// TwinCAT 3 PLC project SFICrane
// ProgramVersion: 3.1.4023.0
// libraries:
//   Tc2_MC2, * (Beckhoff Automation GmbH)
//   Tc2_MC2_Drive, * (Beckhoff Automation GmbH)
//   Tc2_Standard, * (Beckhoff Automation GmbH)
//   Tc2_System, * (Beckhoff Automation GmbH)
//   Tc2_Utilities, * (Beckhoff Automation GmbH)
//   Tc3_Module, * (Beckhoff Automation GmbH)
//   VisuDialogs, * (System)
// project tree:
//   AXIS CONTROL/ G_AXIS1.TcGVL, G_AXIS2.TcGVL, G_AXIS3.TcGVL, G_AXIS4.TcGVL, G_Safety_AXIS4.TcGVL, P_AxisControl.TcPOU, ST_MC_CMD.TcDUT (not stored), ST_MC_ParametersAxis.TcDUT (not stored), ST_MC_Status.TcDUT
//   / GlobalTextList.TcGTLO, MAIN.TcPOU, PlcTask.TcTTO, Visualization Manager.TcVMO (not stored)
//   HMI/ HMI.TcVIS
//   INPUTS/Function Blocks/ FB_AnalogInputScaling.TcPOU (not stored), FB_JoystickInputScaling.TcPOU (not stored)
//   INPUTS/GVL/ G_Inputs.TcGVL (not stored), G_ScalingParameters.TcGVL, G_Sensors.TcGVL
//   INPUTS/ P_Inputs.TcPOU
//   INPUTS/Struct/ ST_AnalogInput.TcDUT, ST_AnalogInputScaling.TcDUT (not stored), ST_AnalogInputStatus.TcDUT (not stored), ST_JoystickInputScaling.TcDUT (not stored), ST_Parameters.TcDUT (not stored)
//   MACHINE CONTROL/ G_MachineControl.TcGVL, P_MachineControl.TcPOU
//   MACHINE CONTROL/KinematicFunctions2d/ cosd.TcPOU (not stored), FB_Forward.TcPOU, FB_Inverse.TcPOU, FB_WireLengthOnCraneFunction.TcPOU, G_InverseKinematics.TcGVL, rt_ceild.TcPOU (not stored), rt_floord.TcPOU (not stored), rt_remd.TcPOU (not stored)
//   OUTPUTS/ G_Outputs.TcGVL, P_Outputs.TcPOU (not stored)
//   StablePlatform/Function Blocks/ FB_AnalogInputScalingPlusMinus.TcPOU, FB_AnalogInputScaling_1.TcPOU, FB_AutoModeControl.TcPOU, FB_Clock.TcPOU, FB_CylinderMotionControl.TcPOU, FB_JoystickInputScaling_1.TcPOU (not stored), FB_LowpassFilter.TcPOU, FB_RampMotionGenerator.TcPOU, FB_ValveOutput.TcPOU (not stored), FB_WaveMotionGenerator.TcPOU, FB_WaveMotionGenerator_1.TcPOU
//   StablePlatform/Functions/ fPlatformAngleTheta1.TcPOU, F_deg2rad.TcPOU, F_rad2deg.TcPOU, F_PlatformAnglePos2CylPos.TcPOU, F_PlatformAngleVel2CylVel.TcPOU
//   StablePlatform/GVL/ G_StablePlatformIO.TcGVL, G_StablePlatformParameters.TcGVL, G_StablePlatformScaledIO.TcGVL
//   StablePlatform/ P_StablePlatform.TcPOU, StablePlatform.TcVIS
//   StablePlatform/Struct/ ST_AnalogInputScaling_1.TcDUT (not stored), ST_JoystickInputScaling_1.TcDUT (not stored), ST_ValveDeadBand.TcDUT (not stored), ST_ValveOutput.TcDUT (not stored)
// real-time tasks:
//   TASK PlcTask: cycle T#2ms, priority 20, ADS port 350
// motion (NC):
//   TASK NC-Task 1 SAF: cycle T#2ms, priority 4, ADS port 501
//   TASK NC-Task 1 SVB: cycle T#10ms, priority 8, ADS port 511
//   AXIS Axis 1 - Main boom Cylinder (id 1)
//     Velo: SlowManual=20, FastManual=100
//     OtherSettings: AllowMotionCmdToSlave=true
//     encoder EncType=8
//       EncPara: MaxCount=#x0036ee7f
//         SoftEndMinControl: Enable=true, Range=12
//         SoftEndMaxControl: Enable=true, Range=298
//     drive DrvType=9
//       DrvPara: MaxCount=#xffffffff, DriveControlDWord=#x00030000
//         Analog: VeloScale=6, TorqueSetpointScale=10, ScaleFactorActTorque=0.1
//         TimeComp: TaskDelayCycles=1
//     controller CtrType=1
//       CtrPara: PriorControlFactor=1
//         Observer: BandWidth=20
//   AXIS Axis 2 - Slew Motor (id 5)
//     General: UnitName=Degree
//     Dynamic: AccelerationMaximum=55000, DecelerationMaximum=55000, Acceleration=30000, Deceleration=30000, Jerk=55000
//     Velo: SlowManual=200, FastManual=1000, Maximum=6000
//     OtherSettings: AllowMotionCmdToSlave=true, PulseDistancePos=100, PulseDistanceNeg=100
//     encoder EncType=8
//       EncPara: MaxCount=#xffffffff
//         SoftEndMinControl: Enable=true, Range=-32870
//         SoftEndMaxControl: Enable=true, Range=32800
//     drive DrvType=9
//       DrvPara: MaxCount=#xffffffff, DriveControlDWord=#x00030000
//         Analog: VeloReferenz=5000, VeloScale=6, TorqueSetpointScale=10, ScaleFactorActTorque=0.1
//         TimeComp: TaskDelayCycles=1
//     controller CtrType=1
//       CtrPara: PriorControlFactor=1
//         PosDiffControl: Range=20
//         Observer: BandWidth=20
//   AXIS Axis 3 - Knuckle boom Cylinder (id 3)
//     Velo: SlowManual=20, FastManual=100
//     OtherSettings: AllowMotionCmdToSlave=true
//     encoder EncType=8
//       EncPara: MaxCount=#x0036ee7f
//         SoftEndMinControl: Enable=true, Range=12
//         SoftEndMaxControl: Enable=true, Range=248
//     drive DrvType=9
//       DrvPara: MaxCount=#xffffffff, DriveControlDWord=#x00030000
//         Analog: VeloScale=6, TorqueSetpointScale=10, ScaleFactorActTorque=0.1
//         TimeComp: TaskDelayCycles=1
//     controller CtrType=1
//       CtrPara: PriorControlFactor=1
//         Observer: BandWidth=20
//   AXIS Axis 4 - Winch Motor (id 4)
//     General: UnitName=°
//     Dynamic: AccelerationMaximum=48322.755, DecelerationMaximum=48322.755, Acceleration=8053.79, Deceleration=8053.79, Jerk=24161.4
//     Velo: RefSearch=53.69195, RefSync=53.69195, SlowManual=268.45975, FastManual=1610.7585, Fast=5369.195
//     OtherSettings: AllowMotionCmdToSlave=true
//     encoder EncType=19
//       EncPara: ScaleFactorNumerator=60, ScaleFactorDenominator=1048576, MaxCount=#xffffffff
//     drive DrvType=16
//       DrvPara: MaxCount=#xffffffff, DriveControlDWord=#x00020000
//         Analog: VeloReferenz=5906.1145, VeloScale=32, TorqueSetpointScale=10, ScaleFactorActTorque=0.1
//         TimeComp: TaskDelayCycles=1
//     controller CtrType=1
//       CtrPara: PriorControlFactor=1
//         PosDiffControl: Enable=false
//         Observer: BandWidth=20
// I/O:
//   DEVICE Device 5 (EtherCAT), AmsNetId 5.107.189.26.6.1
//     Term 29 (EK1914) [EK1914, 2 Ch. Safety Input/Output 24V,  TwinSAFE]
//       modules: Module 1 (FSOE), Module 2 (DIO)
//     Drive 17 (IndraDrive MPB16/17) [IndraDrive MPB16/17]
//     Drive 22 (IndraDrive MPB20/21) [IndraDrive MPB20/21]
//     Drive 23 (IndraDrive MPB20/21) [IndraDrive MPB20/21]
//     Box 24 (AMI8000-0100) [AMI8000-0100 Servo motor 48 V DC, TwinSAFE]
//       modules: Module 1 (SAFETY)
//       startup 32785:21 := 0E01 // DRV Motor Settings / Commutation offset
//       startup 32786:19 := 0000 // DRV Brake Settings / Emergency application timeout
//       startup 32784:51 := 0A00 // DRV Amplifier Settings / Stand still window
//       startup 32784:19 := 2700 // DRV Amplifier Settings / Current loop proportional gain
//       startup 32784:18 := 1300 // DRV Amplifier Settings / Current loop integral time
//       startup 32784:21 := 1F010000 // DRV Amplifier Settings / Velocity loop proportional gain
//       startup 32784:20 := 96000000 // DRV Amplifier Settings / Velocity loop integral time
//   DEVICE Device 1 (EtherCAT), AmsNetId 5.107.189.26.2.1
//     Term 18 (EK1200) [EK1200-5000 EtherCAT Power supply (2A E-Bus)]
//       Term 20 (EL6910) [EL6910, TwinSAFE PLC]
//       Term 21 (EL1904) [EL1904, 4 Ch. Safety Input 24V, TwinSAFE]
//         modules: Module 1 (FSOES)
//       Term 25 (EL2008-0015) [EL2008-0015 8Ch. Dig. Output 24V DC, 0.35A, not short-circuit proof]
//       Term 26 (EK1110) [EK1110 EtherCAT extension]
//     Term 1 (EK1100) [EK1100 EtherCAT Coupler (2A E-Bus)]
//       Term 30 (EL3102) [EL3102 2Ch. Ana. Input +/-10V, Diff.]
//       Term 31 (EL3064) [EL3064 4Ch. Ana. Input 0-10V]
//       Term 32 (EL3124) [EL3124 4Ch. Ana. Input 4-20mA Diff.]
//       Term 33 (EL3154) [EL3154 4Ch. Ana. Input 4-20mA]
//       Term 34 (EL4122) [EL4122 2Ch. Ana. Output  4-20mA, 16bit]
//       Term 35 (EL3002) [EL3002 2Ch. Ana. Input +/-10V]
//       Term 36 (EL4132) [EL4132 2Ch. Ana. Output +/-10V, 16bit]
//       Term 37 (EL1859) [EL1859 8Ch. Dig. Input 24V, 3ms, 8Ch. Dig. Output 24V, 0.5A]
//       Term 35 (EL9011) [EL9011 End Terminal]
//     Term 27 (EK1818) [EK1818 EtherCAT IO-Coupler  (1A E-Bus, 8 Ch. Dig. In, 3ms, 4 Ch. Dig. Out 24V, 0,5A)]
//       Term 28 (EL3255) [EL3255 5Ch. potentiometer measurement with sensor supply]
//       Term 34 (EL9011) [EL9011 End Terminal]
// variable links:
//   Device 1 (EtherCAT) <-> Device 1 (EtherCAT)/Term 18 (EK1200)/Term 20 (EL6910)
//     Term 18 (EK1200)/Term 21 (EL1904)/Module 1 (FSOES)/TxPDO/FSOE <-> ConnectionOutputs/Message_4 RxPDO
//   Device 1 (EtherCAT) <-> Device 1 (EtherCAT)/Term 18 (EK1200)/Term 21 (EL1904)
//     Term 18 (EK1200)/Term 20 (EL6910)/ConnectionInputs/Message_4 TxPDO <-> Module 1 (FSOES)/RxPDO/FSOE
//   Device 1 (EtherCAT) <-> Device 5 (EtherCAT)/Box 24 (AMI8000-0100)
//     Term 18 (EK1200)/Term 20 (EL6910)/ConnectionInputs/Message_3 TxPDO <-> Module 1 (SAFETY)/SAFETY FSoE Connection 1 Receive Message/FSOE
//   Device 1 (EtherCAT) <-> Device 5 (EtherCAT)/Term 29 (EK1914)
//     Term 18 (EK1200)/Term 20 (EL6910)/ConnectionInputs/Message_5 TxPDO <-> Module 1 (FSOE)/Outputs/FSOE
//   Device 5 (EtherCAT) <-> Device 1 (EtherCAT)/Term 18 (EK1200)/Term 20 (EL6910)
//     Box 24 (AMI8000-0100)/Module 1 (SAFETY)/SAFETY FSoE Connection 1 Send Message/FSOE <-> ConnectionOutputs/Message_3 RxPDO
//     Term 29 (EK1914)/Module 1 (FSOE)/Inputs/FSOE <-> ConnectionOutputs/Message_5 RxPDO
//   NC-Task 1 SAF/Axes/Axis 1 - Main boom Cylinder <-> Device 5 (EtherCAT)/Drive 17 (IndraDrive MPB16/17)
//     Drive/Inputs/In/nDcOutputTime <-> InfoData/DcOutputShift
//     Drive/Inputs/In/nState1 <-> AT/Drive status word @bit 8
//     Drive/Inputs/In/nState2 <-> AT/Drive status word
//     Drive/Inputs/In/nState4 @bit 1 <-> WcState/InputToggle
//     Drive/Inputs/In/nState4 <-> WcState/WcState
//     Drive/Outputs/Out/nCtrl1 <-> MDT/Master control word @bit 8
//     Drive/Outputs/Out/nDataOut1 <-> MDT/Position command value
//     Enc/Inputs/In/nDataIn1 <-> AT/Position feedback value 1
//     Enc/Inputs/In/nDcInputTime <-> InfoData/DcInputShift
//     Enc/Inputs/In/nState4 @bit 1 <-> WcState/InputToggle
//     Enc/Inputs/In/nState4 <-> WcState/WcState
//   NC-Task 1 SAF/Axes/Axis 2 - Slew Motor <-> Device 5 (EtherCAT)/Drive 22 (IndraDrive MPB20/21)
//     Drive/Inputs/In/nDcOutputTime <-> InfoData/DcOutputShift
//     Drive/Inputs/In/nState1 <-> AT/Drive status word @bit 8
//     Drive/Inputs/In/nState2 <-> AT/Drive status word
//     Drive/Inputs/In/nState4 @bit 1 <-> WcState/InputToggle
//     Drive/Inputs/In/nState4 <-> WcState/WcState
//     Drive/Outputs/Out/nCtrl1 <-> MDT/Master control word @bit 8
//     Drive/Outputs/Out/nDataOut1 <-> MDT/Position command value
//     Enc/Inputs/In/nDataIn1 <-> AT/Position feedback value 1
//     Enc/Inputs/In/nDcInputTime <-> InfoData/DcInputShift
//     Enc/Inputs/In/nState4 @bit 1 <-> WcState/InputToggle
//     Enc/Inputs/In/nState4 <-> WcState/WcState
//   NC-Task 1 SAF/Axes/Axis 3 - Knuckle boom Cylinder <-> Device 5 (EtherCAT)/Drive 23 (IndraDrive MPB20/21)
//     Drive/Inputs/In/nDcOutputTime <-> InfoData/DcOutputShift
//     Drive/Inputs/In/nState1 <-> AT/Drive status word @bit 8
//     Drive/Inputs/In/nState2 <-> AT/Drive status word
//     Drive/Inputs/In/nState4 @bit 1 <-> WcState/InputToggle
//     Drive/Inputs/In/nState4 <-> WcState/WcState
//     Drive/Outputs/Out/nCtrl1 <-> MDT/Master control word @bit 8
//     Drive/Outputs/Out/nDataOut1 <-> MDT/Position command value
//     Enc/Inputs/In/nDataIn1 <-> AT/Position feedback value 1
//     Enc/Inputs/In/nDcInputTime <-> InfoData/DcInputShift
//     Enc/Inputs/In/nState4 @bit 1 <-> WcState/InputToggle
//     Enc/Inputs/In/nState4 <-> WcState/WcState
//   NC-Task 1 SAF/Axes/Axis 4 - Winch Motor <-> Device 5 (EtherCAT)/Box 24 (AMI8000-0100)
//     Drive/Inputs/In/nDataIn1 <-> DRV Following error actual value/Following error actual value
//     Drive/Inputs/In/nDcOutputTime <-> InfoData/DcOutputShift
//     Drive/Inputs/In/nState1 <-> DRV Statusword/Statusword
//     Drive/Inputs/In/nState2 <-> DRV Statusword/Statusword @bit 8
//     Drive/Inputs/In/nState4 @bit 1 <-> WcState/InputToggle
//     Drive/Inputs/In/nState4 <-> WcState/WcState
//     Drive/Outputs/Out/nCtrl1 <-> DRV Controlword/Controlword
//     Drive/Outputs/Out/nCtrl2 <-> DRV Controlword/Controlword @bit 8
//     Drive/Outputs/Out/nDataOut1 <-> DRV Target position/Target position
//     Drive/Outputs/Out/nDataOut2 <-> DRV Target velocity/Target velocity
//     Enc/Inputs/In/nDataIn1 <-> FB Position/Position
//     Enc/Inputs/In/nDcInputTime <-> InfoData/DcInputShift
//     Enc/Inputs/In/nState4 @bit 1 <-> WcState/InputToggle
//     Enc/Inputs/In/nState4 <-> WcState/WcState
//   SFICrane/SFICrane Instance <-> Device 1 (EtherCAT)/Term 1 (EK1100)/Term 31 (EL3064)
//     PlcTask Inputs/G_StablePlatformIO.npA <-> AI Standard Channel 1/Value
//     PlcTask Inputs/G_StablePlatformIO.npB <-> AI Standard Channel 2/Value
//     PlcTask Inputs/G_StablePlatformIO.npS <-> AI Standard Channel 3/Value
//   SFICrane/SFICrane Instance <-> Device 1 (EtherCAT)/Term 1 (EK1100)/Term 33 (EL3154)
//     PlcTask Inputs/G_StablePlatformIO.nSVFeedback <-> AI Standard Channel 1/Value
//   SFICrane/SFICrane Instance <-> Device 1 (EtherCAT)/Term 1 (EK1100)/Term 34 (EL4122)
//     PlcTask Outputs/G_StablePlatformIO.nSVControlSignal <-> Channel 1/Output
//   SFICrane/SFICrane Instance <-> Device 1 (EtherCAT)/Term 1 (EK1100)/Term 35 (EL3002)
//     PlcTask Inputs/G_StablePlatformIO.nPistonPosition <-> AI Standard Channel 1/Value
//     PlcTask Inputs/G_StablePlatformIO.nPistonVelocity <-> AI Standard Channel 2/Value
//   SFICrane/SFICrane Instance <-> Device 1 (EtherCAT)/Term 1 (EK1100)/Term 37 (EL1859)
//     PlcTask Outputs/G_StablePlatformIO.bSVEnable <-> Channel 14/Output
//   SFICrane/SFICrane Instance <-> Device 1 (EtherCAT)/Term 18 (EK1200)/Term 20 (EL6910)
//     PlcTask Inputs/G_Safety_AXIS4.ChA_STO_Active <-> StandardInputs/Standard Out Var 10
//     PlcTask Inputs/G_StablePlatformIO.bEMG_OK <-> StandardInputs/Standard Out Var 12
//     PlcTask Outputs/G_Safety_AXIS4.EMGRestart <-> StandardOutputs/Standard In Var 8
//     PlcTask Outputs/G_Safety_AXIS4.TwinSafeGroupComErrAck <-> StandardOutputs/Standard In Var 1
//     PlcTask Outputs/G_Safety_AXIS4.TwinSafeGroupRunStop <-> StandardOutputs/Standard In Var 2
//   SFICrane/SFICrane Instance <-> Device 1 (EtherCAT)/Term 18 (EK1200)/Term 25 (EL2008-0015)
//     PlcTask Outputs/G_Safety_AXIS4.bWinchMotor24vDisable <-> Channel 1/Output
//   SFICrane/SFICrane Instance <-> Device 1 (EtherCAT)/Term 27 (EK1818)
//     PlcTask Inputs/G_Inputs.bAutoModeSelector <-> Channel 4/Input
//     PlcTask Inputs/G_Inputs.bGreenButton <-> Channel 5/Input
//     PlcTask Inputs/G_Inputs.bJoystickLeftEnable <-> Channel 7/Input
//     PlcTask Inputs/G_Inputs.bJoystickRightEnable <-> Channel 8/Input
//     PlcTask Inputs/G_Inputs.bManualModeSelector <-> Channel 3/Input
//     PlcTask Inputs/G_Inputs.bRedButton <-> Channel 6/Input
//     PlcTask Inputs/G_StablePlatformIO.bModeSwitchOff <-> Channel 2/Input
//     PlcTask Outputs/G_Outputs.bGreenButtonLight <-> Channel 9/Output
//     PlcTask Outputs/G_Outputs.bRedButtonLight <-> Channel 10/Output
//   SFICrane/SFICrane Instance <-> Device 1 (EtherCAT)/Term 27 (EK1818)/Term 28 (EL3255)
//     PlcTask Inputs/G_Inputs.stJoyLX.nValue <-> AI Standard Channel 1/Value
//     PlcTask Inputs/G_Inputs.stJoyLX.stStatus <-> AI Standard Channel 1/Status
//     PlcTask Inputs/G_Inputs.stJoyLY.nValue <-> AI Standard Channel 2/Value
//     PlcTask Inputs/G_Inputs.stJoyLY.stStatus <-> AI Standard Channel 2/Status
//     PlcTask Inputs/G_Inputs.stJoyRX.nValue <-> AI Standard Channel 3/Value
//     PlcTask Inputs/G_Inputs.stJoyRX.stStatus <-> AI Standard Channel 3/Status
//     PlcTask Inputs/G_Inputs.stJoyRY.nValue <-> AI Standard Channel 4/Value
//     PlcTask Inputs/G_Inputs.stJoyRY.stStatus <-> AI Standard Channel 4/Status
//   SFICrane/SFICrane Instance <-> Device 5 (EtherCAT)/Term 29 (EK1914)
//     PlcTask Inputs/G_Inputs.bSafetyRelayRestartButton <-> Module 2 (DIO)/DIO Inputs/Input 0
//     PlcTask Outputs/G_Outputs.bSafetyRelayReset <-> Module 2 (DIO)/DIO Outputs/Output 0
//   SFICrane/SFICrane Instance <-> NC-Task 1 SAF/Axes/Axis 1 - Main boom Cylinder
//     PlcTask Inputs/G_AXIS1.BCAxis.NcToPlc <-> Outputs/ToPlc
//     PlcTask Inputs/G_MachineControl.fStrokeActuatorMain <-> Outputs/ToPlc/ActPos
//     PlcTask Outputs/G_AXIS1.BCAxis.PlcToNc <-> Inputs/FromPlc
//   SFICrane/SFICrane Instance <-> NC-Task 1 SAF/Axes/Axis 2 - Slew Motor
//     PlcTask Inputs/G_AXIS2.SJAxis.NcToPlc <-> Outputs/ToPlc
//     PlcTask Inputs/G_MachineControl.fSlewMotorAngle <-> Outputs/ToPlc/ActPos
//     PlcTask Outputs/G_AXIS2.SJAxis.PlcToNc <-> Inputs/FromPlc
//   SFICrane/SFICrane Instance <-> NC-Task 1 SAF/Axes/Axis 3 - Knuckle boom Cylinder
//     PlcTask Inputs/G_AXIS3.TCAxis.NcToPlc <-> Outputs/ToPlc
//     PlcTask Inputs/G_MachineControl.fStrokeActuatorKnuckle <-> Outputs/ToPlc/ActPos
//     PlcTask Outputs/G_AXIS3.TCAxis.PlcToNc <-> Inputs/FromPlc
//   SFICrane/SFICrane Instance <-> NC-Task 1 SAF/Axes/Axis 4 - Winch Motor
//     PlcTask Inputs/G_AXIS4.WMAxis.NcToPlc <-> Outputs/ToPlc
//     PlcTask Inputs/G_MachineControl.fWinchMotorAngleEncoder <-> Outputs/ToPlc/ActPos
//     PlcTask Outputs/G_AXIS4.WMAxis.PlcToNc <-> Inputs/FromPlc

CONFIGURATION SFICrane
    RESOURCE PLC ON TwinCAT3
        TASK PlcTask(INTERVAL := T#2ms, PRIORITY := 20);
        PROGRAM MAIN WITH PlcTask : MAIN;
    END_RESOURCE
END_CONFIGURATION

// ---- AXIS CONTROL/ST_MC_Status.TcDUT
TYPE ST_MC_Status :
STRUCT
	
Status			: BOOL;
Done			: BOOL;
Busy			: BOOL;
Error			: BOOL;
Active			: BOOL;
CmdAborted		: BOOL;
InVelocity		: BOOL;
ErrorID			: UDINT;
Enabled			: BOOL;

END_STRUCT
END_TYPE

// ---- INPUTS/Struct/ST_AnalogInput.TcDUT
TYPE ST_AnalogInput :
STRUCT
	stStatus AT %I* : ST_AnalogInputStatus;
	nValue AT %I* : INT;
END_STRUCT
END_TYPE

// ---- AXIS CONTROL/G_AXIS1.TcGVL
{attribute 'qualified_only'}
VAR_GLOBAL

//Axis1 Bottom Cylinder 'BC'
BCAxis : AXIS_REF;

//Motion Control Function Block Instant Variable 
fbBC_Reset				: MC_Reset;
fbBC_Power				: MC_Power;
fbBC_Stop				: MC_Stop;
fbBC_MoveVelocity		: MC_MoveVelocity;
fbBC_MoveAbs			: MC_MoveAbsolute;
fbBC_ExtSetDis			: MC_ExtSetPointGenDisable;
fbBC_ExtSetEnab			: MC_ExtSetPointGenEnable;
fbBC_ResetSet			: RS;

//Input: Command
bBC_ResetExe			: BOOL;
bBC_PowerEnCmd			: BOOL;
bBC_PowerEnPositive		: BOOL;
bBC_PowerEnNegative 	: BOOL;
bBC_StopExe				: BOOL;
bBC_MoveAbsExe			: BOOL;
bBC_ExtSetGenDisExe		: BOOL;
bBC_ExtSetGenEnaExe		: BOOL;
bBC_MoveAbsDone			: BOOL;

//Velocity commands structure
stBC_VelCmd				: ST_MC_CMD := (bExe := FALSE, lrVelocity := 100);//, EnuDirection := MC_Positive_Direction); 

//Variables/Parameters
lrBC_PowerOverride		: LREAL;
lrBC_MoveAbsPosition	: LREAL;
lrBC_MoveAbsVelocity	: LREAL;
lrBC_MoveAddPos			: LREAL;

// Status
stBC_Reset				: ST_MC_Status;
stBC_Power				: ST_MC_Status;
stBC_Stop				: ST_MC_Status;
stBC_MoveVelocity		: ST_MC_Status;
stBC_MoveAbs			: ST_MC_Status;
stBC_ExtSetDis			: ST_MC_Status;
stBC_ExtSetEnab			: ST_MC_Status;
stBC_ExtSetFeed			: ST_MC_Status;

END_VAR

// ---- AXIS CONTROL/G_AXIS2.TcGVL
{attribute 'qualified_only'}
VAR_GLOBAL

//Axis2 Slew Joint 'SJ'
SJAxis : AXIS_REF;

//Motion Control Function Block Instant Variable 
fbSJ_Reset				: MC_Reset;
fbSJ_Power				: MC_Power;
fbSJ_MoveVelocity		: MC_MoveVelocity;
fbSJ_Stop				: MC_Stop;

//Input: Command
bSJ_ResetExe			: BOOL;
bSJ_PowerEnCmd			: BOOL;
bSJ_PowerEnPositive		: BOOL;
bSJ_PowerEnNegative 	: BOOL;
bSJ_StopExe				: BOOL;

//Velocity commands structure
stSJ_VelCmd				: ST_MC_CMD := (bExe := FALSE, lrVelocity := 500, EnuDirection := MC_Positive_Direction); 

//Variables/Parameters
lrSJ_PowerOverride		: LREAL;

// Status
stSJ_Reset				: ST_MC_Status;
stSJ_Power				: ST_MC_Status;
stSJ_MoveVelocity		: ST_MC_Status;
stSJ_Stop				: ST_MC_Status;

END_VAR

// ---- AXIS CONTROL/G_AXIS3.TcGVL
{attribute 'qualified_only'}
VAR_GLOBAL

//Axis3 Top Cylinder 'TC'
TCAxis : AXIS_REF;

//Motion Control Function Block Instant Variable 
fbTC_Reset				: MC_Reset;
fbTC_Power				: MC_Power;
fbTC_MoveVelocity		: MC_MoveVelocity;
fbTC_Stop				: MC_Stop;
fbTC_MoveAbs			: MC_MoveAbsolute;
fbTC_ExtSetDis			: MC_ExtSetPointGenDisable;
fbTC_ExtSetEnab			: MC_ExtSetPointGenEnable;
fbTC_ResetSet			: RS;

//Input: Command
bTC_ResetExe			: BOOL;
bTC_PowerEnCmd			: BOOL;
bTC_PowerEnPositive		: BOOL;
bTC_PowerEnNegative 	: BOOL;
bTC_StopExe				: BOOL;
bTC_MoveAbsExe			: BOOL;
bTC_ExtSetGenDisExe		: BOOL;
bTC_ExtSetGenEnaExe		: BOOL;
bTC_MoveAbsDone			: BOOL;

//Velocity commands structure
stTC_VelCmd				: ST_MC_CMD := (bExe := FALSE, lrVelocity := 100, EnuDirection := MC_Positive_Direction); 

//Variables/Parameters
lrTC_PowerOverride		: LREAL;
lrTC_MoveAbsPosition	: LREAL;
lrTC_MoveAbsVelocity	: LREAL;
lrTC_MoveAddPos			: LREAL;

// Status
stTC_Reset				: ST_MC_Status;
stTC_Power				: ST_MC_Status;
stTC_MoveVelocity		: ST_MC_Status;
stTC_Stop				: ST_MC_Status;
stTC_MoveAbs			: ST_MC_Status;
stTC_ExtSetDis			: ST_MC_Status;
stTC_ExtSetEnab			: ST_MC_Status;
stTC_ExtSetFeed			: ST_MC_Status;

END_VAR

// ---- AXIS CONTROL/G_AXIS4.TcGVL
{attribute 'qualified_only'}
VAR_GLOBAL

//Axis4 Winch Motor 'WM'
WMAxis : AXIS_REF;

//Motion Control Function Block Instant Variable 
fbWM_Reset				: MC_Reset;
fbWM_Power				: MC_Power;
fbWM_MoveVelocity		: MC_MoveVelocity;
fbWM_Stop				: MC_Stop;
fbWM_MoveAbs			: MC_MoveAbsolute;
fbWM_ExtSetDis			: MC_ExtSetPointGenDisable;
fbWM_ExtSetEnab			: MC_ExtSetPointGenEnable;
fbWM_ResetSet			: RS;

//Input: Command
bWM_ResetExe			: BOOL;
bWM_PowerEnCmd			: BOOL;
bWM_PowerEnPositive		: BOOL;
bWM_PowerEnNegative 	: BOOL;
bWM_StopExe				: BOOL;
bWM_MoveAbsExe			: BOOL;
bWM_ExtSetGenDisExe		: BOOL;
bWM_ExtSetGenEnaExe		: BOOL;
bWM_MoveAbsDone			: BOOL;

//Velocity commands structure
stWM_VelCmd				: ST_MC_CMD := (bExe := FALSE, lrVelocity := 1000, EnuDirection := MC_Positive_Direction); 

//Variables/Parameters
lrWM_PowerOverride		: LREAL;
lrWM_MoveAbsPosition	: LREAL;
lrWM_MoveAbsVelocity	: LREAL;
lrWM_MoveAddPos			: LREAL;
lrWM_MoveSetPointVel	: LREAL;

//Direction
EnuMoveVelDirection		: MC_Direction;

// Status
stWM_Reset				: ST_MC_Status;
stWM_Power				: ST_MC_Status;
stWM_MoveVelocity		: ST_MC_Status;
stWM_Stop				: ST_MC_Status;
stWM_MoveAbs			: ST_MC_Status;
stWM_ExtSetDis			: ST_MC_Status;
stWM_ExtSetEnab			: ST_MC_Status;
stWM_ExtSetFeed			: ST_MC_Status;

END_VAR

// ---- AXIS CONTROL/G_Safety_AXIS4.TcGVL
{attribute 'qualified_only'}
VAR_GLOBAL
	
	bWinchMotor24vDisable 		AT %Q* : BOOL;
	TwinSafeGroupComErrAck 		AT %Q* : BOOL; 
	TwinSafeGroupRunStop 		AT %Q* : BOOL := FALSE; 
	ChA_STO_Enable 				AT %Q* : BOOL;
	ChA_STO_Active 				AT %I* : BOOL;  
	EMGRestart 					AT %Q* : BOOL; 
END_VAR

// ---- INPUTS/GVL/G_ScalingParameters.TcGVL
{attribute 'qualified_only'}
VAR_GLOBAL
	stParam : ST_Parameters;
END_VAR

// ---- INPUTS/GVL/G_Sensors.TcGVL
{attribute 'qualified_only'}
VAR_GLOBAL
	fJoystickLeftNormalizedY 		: LREAL;
	fJoystickLeftNormalizedX 		: LREAL;
	
	fJoystickRightNormalizedY 		: LREAL;
	fJoystickRightNormalizedX 		: LREAL;
	
	MCDirectionAxis1 : MC_Direction;
	MCDirectionAxis2 : MC_Direction;
	MCDirectionAxis3 : MC_Direction;
	MCDirectionAxis4 : MC_Direction;
	
		
END_VAR

// ---- MACHINE CONTROL/G_MachineControl.TcGVL
{attribute 'qualified_only'}
VAR_GLOBAL
	//Mode selector booleans
	bManualMode 			: BOOL;
	bAutoMode 				: BOOL;
	
	//Time variables
	fSampleTime				: LREAL := 0.002;
	fTimeSinceStart			: LREAL := 0.0;
	
	//Actuator position data
	fStrokeActuatorMain 	AT %I* : LREAL;
	fStrokeActuatorKnuckle 	AT %I* : LREAL;
	fSlewMotorAngle			AT %I* : LREAL;
	fWinchMotorAngleEncoder		AT %I* : LREAL;	
	fWinchAngle				: LREAL;
	fWinchMotorAngleRefDeg	: LREAL;
	
	//Positions from forward kinematics
	fCraneForwardX 			: LREAL;
	fCraneForwardY 			: LREAL;
	fTheta3Forward			: LREAL;
	fTheta4Forward			: LREAL;
	
	//Working parameters crane
	fWireLengthOnCrane		: LREAL;
	fPayloadHeightIni		: LREAL := 0.0;
	fWinchPitchRadiusLayer1 : LREAL := 0.0716;
	fWinchPitchRadiusLayer2 : LREAL := 0.0731;
	fWinchGearRatio 		: LREAL := 32;
	fWinchMotorAngleAbsRef	: LREAL;
	
	//Encoder values 
	fEncoderValue0Turns		: LREAL := 0.0;
	fEncoderValue5Turns		: LREAL := 0.0;
	fEncoderValueLayer2		: LREAL := 23666.0;
	fEncoderValueStartAuto	: LREAL;
	fTooltipYAutoStart		: LREAL;
	fRefPosPayloadAutoStart	: LREAL;
	fWinchMotorAngleRelRef	: LREAL;
	
	

END_VAR

// ---- MACHINE CONTROL/KinematicFunctions2d/G_InverseKinematics.TcGVL
{attribute 'qualified_only'}
VAR_GLOBAL
	fTooltipXCoordGlobalIni: LREAL := 2.8;
	fTooltipYCoordGlobalIni: LREAL := 2.2;
	
	fTheta1 : LREAL := 0;
	fAngleMainArmInverse :	LREAL;
	fAngleKnuckleArmInverse : LREAL;
	fStrokeActuatorMainInverse : LREAL;
	fStrokeActuatorKnuckleInverse : LREAL;
END_VAR

// ---- OUTPUTS/G_Outputs.TcGVL
{attribute 'qualified_only'}
VAR_GLOBAL
	// PLC Rack
	
	// RIO Rack
	// Digital Outputs
	bGreenButtonLight 			AT %Q* : BOOL;
	bRedButtonLight 			AT %Q* : BOOL;
	// Analog Outputs
	//stWinchValveOutput 		: ST_ValveOutput;
	//stCylValveOutput 			: ST_ValveOutput;
	bSafetyRelayReset		 	AT %Q* : BOOL;
END_VAR

// ---- StablePlatform/GVL/G_StablePlatformIO.TcGVL
{attribute 'qualified_only'}
VAR_GLOBAL
	bSVEnable AT %Q* : BOOL; 
	nSVControlSignal AT %Q* : INT; 
	//fJoyLeftX AT %I* : INT; 
	
	//bJoyLeftPushButton AT %I* : BOOL; 
	
	npA AT %I* : INT;
	npB AT %I* : INT;
	npS AT %I* : INT;
	
	nSVFeedback AT %I* : INT;
	
	bModeSwitchOff AT %I* : BOOL;
	
	nPistonPosition AT %I* : INT;
	nPistonVelocity AT %I* : INT;

	// TwinSAFE	
	bEMG_OK AT %I* : BOOL;
	
	// Visualizer HMI
	bEnable : BOOL;
	bModeSelector : BOOL;
	bManualMode : BOOL;
	bAutoMode : BOOL;
	bActivated : BOOL;
	
	// Stable Control
	bEnableFeedForward 		: BOOL := TRUE;
	fMaxValveFlow_lmin 		: LREAL := 45.0;
	bEnableFeedBackControl	: BOOL := TRUE;
	bEnableIntegralControl	: BOOL := FALSE;
	fProportionalGain		: LREAL := 25.0;
	fIntegralGain			: LREAL := 0.0;
	fMaxPosError_mm			: LREAL := 0.5;
	fCylVelRef_ms			: LREAL;
	fCylPosRef_m			: LREAL;
	fCylPos_m				: LREAL;
	bMotionModeSelector : BOOL;
	bStartMotionGenerator : BOOL;
	bRampMotionFullPeriode : BOOL;
	bRampMotionPos0_deg: LREAL := -2.0; 
	bRampMotionCylVel0_ms : LREAL := 0.0; 
	bRampMotionPositionSP_deg : LREAL := 0;
	bRampMotionVelocitySP_ms : LREAL := 0.025; 
	bRampMotiont0_s : LREAL := 1.0; 
	bRampMotiontRamp_s : LREAL := 1.0; 
	bRampMotiontHoldPos_s : LREAL := 2.0;

	fTime : LREAL;
	fWaveMotionAplitudeTheta0_deg : LREAL := -1.9; 
	WaveMotionFreq_rads : LREAL := 0.5;
	fWaveMotionOmega_degs : LREAL; 
	fWaveMotionTheta_deg : LREAL; 
	fAutoModeControlSignal :LREAL;
	
	fControlSignal : LREAL;
END_VAR

// ---- StablePlatform/GVL/G_StablePlatformParameters.TcGVL
{attribute 'qualified_only'}
VAR_GLOBAL
	stPressureSensorScaling400bar 	: ST_AnalogInputScaling := (fMaxInputValue := 32767.0, fMinInputValue := 0.0, fMaxOutputValue := 400.0, fMinOutputValue := 0.0);
	stJoystickInputScalingX 		: ST_JoystickInputScaling := (fMaxInputValue := 20625.0, fMinInputValue := 11800.0, fNeutralInputValue := 16265, fNeutralDeadband := 100.0, fMaxOutputValue := 1.0, fMinOutputValue := -1.0, fNeutralOutputValue := 0.0);
	stSVValveDeadBand 				: ST_ValveDeadBand := (fPosMax := 29490.0, fPosMin := 20950.0, fNegMin := 18250.0, fNegMax := 9830.0);
	stSVFeedbackScaling 			: ST_AnalogInputScaling := (fMaxInputValue := 32767.0, fMinInputValue := 0.0, fMaxOutputValue := 20.0, fMinOutputValue := 4.0);
	stPistonPos						: ST_AnalogInputScaling := (fMaxInputValue := 32767.0, fMinInputValue := -32767.0, fMaxOutputValue := 0.5, fMinOutputValue := 0.0);
	stPistonVel						: ST_AnalogInputScaling := (fMaxInputValue := 32767.0, fMinInputValue := -32767.0, fMaxOutputValue := 0.2, fMinOutputValue := -0.2);
	fMinLengthPlatformCylinder		: LREAL := 0.878;
	fCylLengthZeroAngle				: LREAL := 1.142;
	fLengthToCylinder				: LREAL := 0.500;
	fOffsetAngleDeg 				: LREAL := 55.4;
	fOffsetAngleRad					: LREAL := Tc2_Utilities.DEG_TO_RAD(fOffsetAngleDeg);
	fLengthA						: LREAL := 0.513; //Length from platform bearing to cylinder upper mount
	fLengthC						: LREAL := 1.353; //Length from platform bearing to cylinder lower mount
	fAngleOffsetDeg 				: LREAL := 0.0;
	fMaxControlSignal				: LREAL := 0.2; 
	fCutoffFreq 					: LREAL := 0.1;
	fDamping 						: LREAL := 0.707106781186547;
END_VAR

// ---- StablePlatform/GVL/G_StablePlatformScaledIO.TcGVL
{attribute 'qualified_only'}
VAR_GLOBAL
	bpA : LREAL; // 0..400bar
	bpB : LREAL; // 0..400bar
	bpS : LREAL; // 0..400bar
	fSVFeedback : LREAL; // 4..20 mA  | 0 = fault/off
	fJoystickNormalizedX : LREAL; // -1..0..1
	fPistonPosition : LREAL; //Piston position in meters
	fPistionPosFiltered : LREAL;
	fPistonVelocity : LREAL; //Piston velocity in meters/second
	fPlatformAngle	: LREAL; //Platform angle theta1 in radians
	fPlatformAngleDeg : LREAL;
END_VAR

// ---- MAIN.TcPOU
PROGRAM MAIN

VAR

END_VAR

P_Inputs();
P_MachineControl();
P_AxisControl();
P_Outputs();
P_StablePlatform();

END_PROGRAM

// ---- INPUTS/P_Inputs.TcPOU
PROGRAM P_Inputs
VAR
	fbJoystickLeftVert 					: FB_JoystickInputScaling;
	fbJoystickLeftHor 					: FB_JoystickInputScaling;
	
	fbJoystickRightVert 				: FB_JoystickInputScaling;
	fbJoystickRightHor 					: FB_JoystickInputScaling;
	
	bEnableJoystick : BOOL;
		
END_VAR

bEnableJoystick := NOT(G_StablePlatformIO.bManualMode);

fbJoystickLeftVert(
	bEnable := bEnableJoystick,
	nRawInput := G_Inputs.stJoyLY.nValue,
	stJoystickInputScaling := G_ScalingParameters.stParam.stJoystickInputScalingLeftY,
	fNormalizedOutput => G_Sensors.fJoystickLeftNormalizedY
);

IF G_Sensors.fJoystickLeftNormalizedY < 0 THEN
	G_Sensors.MCDirectionAxis3 := MC_Negative_Direction;
ELSIF G_Sensors.fJoystickLeftNormalizedY > 0 THEN
	G_Sensors.MCDirectionAxis3 := MC_Positive_Direction;	
END_IF

fbJoystickLeftHor(
	bEnable := bEnableJoystick,
	nRawInput := G_Inputs.stJoyLX.nValue,
	stJoystickInputScaling := G_ScalingParameters.stParam.stJoystickInputScalingLeftX,
	fNormalizedOutput => G_Sensors.fJoystickLeftNormalizedX
);

IF G_Sensors.fJoystickLeftNormalizedX < 0 THEN
	G_Sensors.MCDirectionAxis1 := MC_Positive_Direction;
ELSIF G_Sensors.fJoystickLeftNormalizedX > 0 THEN
	G_Sensors.MCDirectionAxis1 := MC_Negative_Direction;	
END_IF


fbJoystickRightVert(
	bEnable := bEnableJoystick,
	nRawInput := G_Inputs.stJoyRY.nValue,
	stJoystickInputScaling := G_ScalingParameters.stParam.stJoystickInputScalingRightY,
	fNormalizedOutput => G_Sensors.fJoystickRightNormalizedY
);

IF G_Sensors.fJoystickRightNormalizedY < 0 THEN
	G_Sensors.MCDirectionAxis4 := MC_Negative_Direction;
ELSIF G_Sensors.fJoystickRightNormalizedY > 0 THEN
	G_Sensors.MCDirectionAxis4 := MC_Positive_Direction;	
END_IF



fbJoystickRightHor(
	bEnable := bEnableJoystick,
	nRawInput := G_Inputs.stJoyRX.nValue,
	stJoystickInputScaling := G_ScalingParameters.stParam.stJoystickInputScalingRightX,
	fNormalizedOutput => G_Sensors.fJoystickRightNormalizedX
);

IF G_Sensors.fJoystickRightNormalizedX < 0 THEN
	G_Sensors.MCDirectionAxis2 := MC_Positive_Direction;
ELSIF G_Sensors.fJoystickRightNormalizedX > 0 THEN
	G_Sensors.MCDirectionAxis2 := MC_Negative_Direction;	
END_IF

END_PROGRAM

// ---- MACHINE CONTROL/P_MachineControl.TcPOU
PROGRAM P_MachineControl
VAR
	fbInverse					: FB_Inverse;
	fbForward					: FB_Forward;
	fbWireLengthOnCrane			: FB_WireLengthOnCraneFunction;
	fRefPosX					: LREAL := G_InverseKinematics.fTooltipXCoordGlobalIni;
	fRefPosY					: LREAL := G_InverseKinematics.fTooltipYCoordGlobalIni;	
	fRefPosPayload				: LREAL := G_MachineControl.fPayloadHeightIni;
	fWireLengthOutAutoStart		: LREAL;
	fWireLengthOut				: LREAL;
	fWireLengthOnCraneAutoStart	: LREAL;
	fWinchPitchRadius			: LREAL;
	fThetaWinch					: LREAL;
	bStartWave					: BOOL;
			
	
	
END_VAR

G_MachineControl.bManualMode := G_Inputs.bManualModeSelector;
G_MachineControl.bAutoMode := G_Inputs.bAutoModeSelector;
G_Safety_AXIS4.ChA_STO_Enable := G_Inputs.bManualModeSelector OR G_Inputs.bAutoModeSelector;

IF G_Inputs.bAutoModeSelector THEN
fRefPosX := fRefPosX + G_Sensors.fJoystickLeftNormalizedX*-0.0005;
fRefPosY := fRefPosY + G_Sensors.fJoystickLeftNormalizedY*0.0005;
fRefPosPayload := fRefPosPayload + G_Sensors.fJoystickRightNormalizedY*0.0002;
END_IF

bStartWave := NOT G_Inputs.bRedButton; //Red button is inverted, i.e. is active when not pushed

//Wave function used for testing
IF bStartWave THEN
	//Clock
	G_MachineControl.fTimeSinceStart := G_MachineControl.fTimeSinceStart + G_MachineControl.fSampleTime;
	G_InverseKinematics.fTheta1 := 0.012*SIN(2.5*G_MachineControl.fTimeSinceStart);
END_IF

(*
IF bStartWave THEN
	//Clock
	G_Work.fTimeSinceStart := G_Work.fTimeSinceStart + G_Work.fSampleTime;
	GVL_InverseKinematics.fTheta1 := G_StablePlatformParameters.fPlatformAngle;
END_IF
*)

fbInverse(
	fPtXd := fRefPosX, 
	fPtYd := fRefPosY, 
	//fTheta1 := G_InverseKinematics.fTheta1,
	fTheta1 := G_StablePlatformScaledIO.fPlatformAngleDeg*(PI/180),
	
	fTheta3 => G_InverseKinematics.fAngleMainArmInverse, 
	fTheta4 => G_InverseKinematics.fAngleKnuckleArmInverse,
	fStrokeActuatorMain => G_InverseKinematics.fStrokeActuatorMainInverse,
	fStrokeActuatorKnuckle => G_InverseKinematics.fStrokeActuatorKnuckleInverse,	
);

fbForward(
	fTheta1 := G_StablePlatformScaledIO.fPlatformAngle,
	fStrokeActuatorMain := (G_MachineControl.fStrokeActuatorMain+11),
	fStrokeActuatorKnuckle := (G_MachineControl.fStrokeActuatorKnuckle-7),
	x => G_MachineControl.fCraneForwardX,
	y => G_MachineControl.fCraneForwardY, 
	fTheta3 => G_MachineControl.fTheta3Forward,
	fTheta4 => G_MachineControl.fTheta4Forward,
);

fbWireLengthOnCrane(
	fTheta3 := G_MachineControl.fTheta3Forward,
	fTheta4 := G_MachineControl.fTheta4Forward,
	wireLengthOnCrane => G_MachineControl.fWireLengthOnCrane,
);

IF NOT (G_Inputs.bAutoModeSelector AND G_AXIS1.bBC_MoveAbsDone AND G_AXIS3.bTC_MoveAbsDone) THEN
	G_MachineControl.fEncoderValueStartAuto := G_MachineControl.fWinchMotorAngleEncoder;
	G_MachineControl.fRefPosPayloadAutoStart := G_MachineControl.fPayloadHeightIni;
	G_MachineControl.fTooltipYAutoStart := G_MachineControl.fCraneForwardY;	
	G_MachineControl.fWinchMotorAngleRelRef := G_MachineControl.fWinchMotorAngleRefDeg;
	fWireLengthOnCraneAutoStart := G_MachineControl.fWireLengthOnCrane;
END_IF

//fWireLengthOutAutoStart := fWireLengthOnCraneAutoStart + (G_MachineControl.fTooltipYAutoStart - G_MachineControl.fRefPosPayloadAutoStart);
fWireLengthOut := G_MachineControl.fWireLengthOnCrane + (G_MachineControl.fCraneForwardY - fRefPosPayload);


IF G_MachineControl.fWinchMotorAngleEncoder > G_MachineControl.fEncoderValueLayer2 THEN
	fWinchPitchRadius := G_MachineControl.fWinchPitchRadiusLayer2;
ELSE
	fWinchPitchRadius := G_MachineControl.fWinchPitchRadiusLayer1;
END_IF

fThetaWinch := (fWireLengthOut / fWinchPitchRadius);
G_MachineControl.fWinchMotorAngleRefDeg := fThetaWinch*G_MachineControl.fWinchGearRatio*180/PI;

IF NOT (G_Inputs.bAutoModeSelector AND G_AXIS1.bBC_MoveAbsDone AND G_AXIS3.bTC_MoveAbsDone) THEN
	G_MachineControl.fEncoderValueStartAuto := G_MachineControl.fWinchMotorAngleEncoder;
	
	G_MachineControl.fWinchMotorAngleRelRef := G_MachineControl.fWinchMotorAngleRefDeg;
END_IF

G_MachineControl.fWinchMotorAngleAbsRef := G_MachineControl.fEncoderValueStartAuto + G_MachineControl.fWinchMotorAngleRelRef - G_MachineControl.fWinchMotorAngleRefDeg;

END_PROGRAM

// ---- MACHINE CONTROL/KinematicFunctions2d/FB_Inverse.TcPOU
FUNCTION_BLOCK FB_Inverse
VAR_INPUT
	fPtXd: LREAL;
	fPtYd: LREAL;
	fTheta1: LREAL;
END_VAR
VAR_OUTPUT
	fStrokeActuatorMain: LREAL;
	fStrokeActuatorKnuckle: LREAL;
	fTheta3: LREAL;
	fTheta4: LREAL;
END_VAR
VAR
	h: LREAL;
	ThetaB: LREAL;
	ThetaB_tmp: LREAL;
	b_a_tmp: LREAL;
	a_tmp: LREAL;
	i0_cosd: cosd;
END_VAR


(* MATLAB Function: '<Root>/Inverse kinematics function' *)
(* clc; close all; clear; *)
(* MATLAB Function 'Inverse kinematics function': '<S1>:1' *)
(* Inputs *)
(* Desired global coordinates *)
(* fPtXd		= 0.75 + 1.5; *)
(* fPtYd		= 1.065 + 0.176; *)

(* %     fPtXd		= 0.75 + 0.716; *)
(* %  	fPtYd		= 1.065 + 0.705; *)
(* Platform constants *)
(* '<S1>:1:14' h0 = 1.0; *)
(* '<S1>:1:15' l0 = 0.75; *)
(* Crane constants *)
(* '<S1>:1:18' h1 = 1.334 + 0.065; *)
(* '<S1>:1:19' lm = 1.5; *)
(* '<S1>:1:20' lk = 1.158; *)
(* Calculate position of a2 as function of Theta1 *)
(* '<S1>:1:23' a2x = l0*cos(fTheta1) + h1*cos(fTheta1 + pi/2); *)
(* '<S1>:1:24' a2y = h0 + l0*sin(fTheta1) + h1*sin(fTheta1 + pi/2); *)
(* '<S1>:1:26' h = sqrt((fPtXd - a2x)^2 + (fPtYd - a2y)^2); *)
a_tmp := fPtXd - ((COS(fTheta1 + 1.5707963267948966) * 1.399) + (0.75 * COS(fTheta1)));
b_a_tmp := fPtYd - (((0.75 * SIN(fTheta1)) + 1.0) + (SIN(fTheta1 + 1.5707963267948966) * 1.399));
h := SQRT((a_tmp * a_tmp) + (b_a_tmp * b_a_tmp));
(* '<S1>:1:27' phi = atan((fPtYd - a2y) / (fPtXd - a2x)); *)
(* Calculate ThetaA and ThetaB *)
(* '<S1>:1:30' ThetaA = acos ((lm^2 + h^2 - lk^2) / (2*lm*h)); *)
(* '<S1>:1:31' ThetaB = acos ((lk^2 + lm^2 - h^2) / (2*lm*lk)); *)
ThetaB_tmp := h * h;
ThetaB := ACOS((3.5909639999999996 - ThetaB_tmp) / 3.4739999999999998);
(* '<S1>:1:33' fTheta3 = ThetaA + phi - fTheta1; *)
fTheta3 := (ACOS(((ThetaB_tmp + 2.25) - 1.3409639999999998) / (3.0 * h)) + ATAN(b_a_tmp / a_tmp)) - fTheta1;
(* '<S1>:1:34' fTheta4 = ThetaB - pi/2; *)
(* '<S1>:1:36' fTheta3deg = rad2deg(fTheta3); *)
(* '<S1>:1:37' fTheta4deg = rad2deg(fTheta4); *)
(* Crane constant parameters *)
(* '<S1>:1:40' fLengthP2PMainArm			= lm; *)
(* '<S1>:1:41' fLengthP2PKnuckleArm		= lk; *)
(* '<S1>:1:43' fLengthAMain				= 0.614; *)
(* '<S1>:1:44' fLengthBMain				= 0.571; *)
(* '<S1>:1:45' fMinLengthActuatorMain		= 0.691; *)
(* '<S1>:1:46' fMaxStrokeActuatorMain		= 0.290; *)
(* 0.320; *)
(* '<S1>:1:47' fMinStrokeActuatorMain		= 0.025; *)
(* '<S1>:1:49' fOffsetAngleDegMainAct		= 62.1; *)
(* '<S1>:1:51' fLengthAKnuckle				= 0.767; *)
(* '<S1>:1:52' fLengthBKnuckle				= 0.184; *)
(* '<S1>:1:53' fMinLengthActuatorKnuckle	= 0.633; *)
(* '<S1>:1:54' fMaxStrokeActuatorKnuckle	= 0.220; *)
(* 0.260; *)
(* '<S1>:1:55' fMinStrokeActuatorKnuckle   = 0.025; *)
(* '<S1>:1:57' fOffsetAngleDegKnuckleAct	= 86.3; *)
(* '<S1>:1:60' fAngleMainArmAct			= fTheta3deg + fOffsetAngleDegMainAct; *)
(* '<S1>:1:61' fAngleKnuckleArmAct         = fTheta4deg + fOffsetAngleDegKnuckleAct; *)
(* '<S1>:1:63' fLengthActuatorMain         = sqrt(fLengthAMain^2 + fLengthBMain^2 -(2*fLengthAMain*fLengthBMain*cosd(fAngleMainArmAct))); *)
(* '<S1>:1:64' fStrokeActuatorMain         = fLengthActuatorMain - fMinLengthActuatorMain; *)
a_tmp := (57.295779513082323 * fTheta3) + 62.1;
b_a_tmp := a_tmp;
i0_cosd(x := b_a_tmp);
(* Outport: '<Root>/fStrokeActuatorMain' incorporates:
 *  MATLAB Function: '<Root>/Inverse kinematics function' *)
fStrokeActuatorMain := SQRT(0.70303699999999991 - (0.70118799999999992 * b_a_tmp)) - 0.691;
(* MATLAB Function: '<Root>/Inverse kinematics function' *)
(* '<S1>:1:66' if fStrokeActuatorMain < fMinStrokeActuatorMain *)
b_a_tmp := a_tmp;
i0_cosd(x := b_a_tmp);

IF (SQRT(0.70303699999999991 - (0.70118799999999992 * b_a_tmp)) - 0.691) < 0.025 THEN 
    (* Outport: '<Root>/fStrokeActuatorMain' *)
    (* '<S1>:1:67' fStrokeActuatorMain = fMinStrokeActuatorMain; *)
    fStrokeActuatorMain := 0.025;
END_IF;

(* '<S1>:1:72' fLengthActuatorKnuckle         = sqrt(fLengthAKnuckle^2 + fLengthBKnuckle^2 -(2*fLengthAKnuckle*fLengthBKnuckle*cosd(fAngleKnuckleArmAct))); *)
(* '<S1>:1:73' fStrokeActuatorKnuckle         = fLengthActuatorKnuckle - fMinLengthActuatorKnuckle; *)
a_tmp := ((ThetaB - 1.5707963267948966) * 57.295779513082323) + 86.3;
b_a_tmp := a_tmp;
i0_cosd(x := b_a_tmp);
(* Outport: '<Root>/fStrokeActuatorKnuckle' incorporates:
 *  MATLAB Function: '<Root>/Inverse kinematics function' *)
fStrokeActuatorKnuckle := SQRT(0.62214500000000006 - (0.282256 * b_a_tmp)) - 0.633;
(* MATLAB Function: '<Root>/Inverse kinematics function' *)
(* '<S1>:1:75' if fStrokeActuatorKnuckle < fMinStrokeActuatorKnuckle *)
b_a_tmp := a_tmp;
i0_cosd(x := b_a_tmp);

IF (SQRT(0.62214500000000006 - (0.282256 * b_a_tmp)) - 0.633) < 0.025 THEN 
    (* Outport: '<Root>/fStrokeActuatorKnuckle' *)
    (* '<S1>:1:76' fStrokeActuatorKnuckle = fMinStrokeActuatorKnuckle; *)
    fStrokeActuatorKnuckle := 0.025;
END_IF;

(* Outport: '<Root>/fTheta4' incorporates:
 *  MATLAB Function: '<Root>/Inverse kinematics function' *)
fTheta4 := ThetaB - 1.5707963267948966;

END_FUNCTION_BLOCK

// ---- MACHINE CONTROL/KinematicFunctions2d/FB_Forward.TcPOU
FUNCTION_BLOCK FB_Forward
VAR_INPUT
	fTheta1: LREAL;
	fStrokeActuatorMain: LREAL;
	fStrokeActuatorKnuckle: LREAL;
END_VAR
VAR_OUTPUT
	x: LREAL;
	y: LREAL;
	fTheta3: LREAL;
	fTheta4: LREAL;
END_VAR
VAR
	x_tmp: LREAL;
	x_tmp_0: LREAL;
END_VAR


(* MATLAB Function: '<Root>/Forward kinematics actuator strokes' *)
(* Platform constants *)
(* MATLAB Function 'Forward kinematics actuator strokes': '<S1>:1' *)
(* '<S1>:1:4' fHeightPlatform = 1.402; *)
(* '<S1>:1:5' fHeightPlatformKing = 0.09; *)
(* '<S1>:1:6' fLengthPlatform = 1.30; *)
(* Crane and platform dimensions *)
(* Crane constant parameters *)
(* '<S1>:1:11' fHeightKingSlew             = 0.623; *)
(* '<S1>:1:12' fHeightSlewTop              = 0.711; *)
(* '<S1>:1:13' fLengthMainArm			    = 1.5; *)
(* '<S1>:1:14' fLengthKnuckleArm		    = 1.158; *)
(* '<S1>:1:16' fLengthAMain				= 0.614; *)
(* '<S1>:1:17' fLengthBMain				= 0.571; *)
(* '<S1>:1:18' fMinLengthActuatorMain		= 0.691; *)
(* '<S1>:1:19' fMaxStrokeActuatorMain		= 0.320; *)
(* '<S1>:1:21' fOffsetAngleDegMainAct		= 62.1; *)
(* '<S1>:1:22' fOffsetAngleRadMainAct		= deg2rad(fOffsetAngleDegMainAct); *)
(* '<S1>:1:24' fLengthAKnuckle				= 0.767; *)
(* '<S1>:1:25' fLengthBKnuckle				= 0.184; *)
(* '<S1>:1:26' fMinLengthActuatorKnuckle	= 0.633; *)
(* '<S1>:1:27' fMaxStrokeActuatorKnuckle	= 0.260; *)
(* '<S1>:1:29' fOffsetAngleDegKnuckleAct	= 86.3; *)
(* '<S1>:1:30' fOffsetAngleRadKnuckleAct	= deg2rad(fOffsetAngleDegKnuckleAct); *)
(* Calculating angles for main arm *)
(* '<S1>:1:33' fLengthActuatorMain = fStrokeActuatorMain + fMinLengthActuatorMain; *)
(* '<S1>:1:35' fAngleMainArmAct = acos((fLengthBMain^2 + fLengthAMain^2 - fLengthActuatorMain^2) / (2 * fLengthBMain * fLengthAMain)); *)
(* '<S1>:1:37' fTheta3 = fAngleMainArmAct - fOffsetAngleRadMainAct; *)
fTheta3 := ACOS((0.70303699999999991 - ((fStrokeActuatorMain/1000 + 0.691) * (fStrokeActuatorMain/1000 + 0.691))) / 0.70118799999999992) - 1.0838494654884787;
(* Calculating angles for knuckle arm *)
(* '<S1>:1:40' fLengthActuatorKnuckle = fStrokeActuatorKnuckle + fMinLengthActuatorKnuckle; *)
(* '<S1>:1:42' fAngleKnuckleArmAct = acos((fLengthBKnuckle^2 + fLengthAKnuckle^2 - fLengthActuatorKnuckle^2) / (2 * fLengthBKnuckle * fLengthAKnuckle)); *)
(* '<S1>:1:44' fTheta4 = fAngleKnuckleArmAct - fOffsetAngleRadKnuckleAct; *)
fTheta4 := ACOS((0.62214500000000006 - ((fStrokeActuatorKnuckle/1000 + 0.633) * (fStrokeActuatorKnuckle/1000 + 0.633))) / 0.282256) - 1.5062191444711064;

(* fAngleMainArmAct			= fTheta3deg + fOffsetAngleDegMainAct; *)
(* fAngleKnuckleArmAct         = fTheta4deg + fOffsetAngleDegKnuckleAct; *)

(* fLengthActuatorMain         = sqrt(fLengthAMain^2 + fLengthBMain^2 -(2*fLengthAMain*fLengthBMain*cosd(fAngleMainArmAct))); *)
(* fStrokeActuatorMain         = fLengthActuatorMain - fMinLengthActuatorMain; *)
(* if fStrokeActuatorMain < 0 *)
(* fStrokeActuatorMain = 0; *)
(* elseif fStrokeActuatorMain > fMaxStrokeActuatorMain *)
(* fMaxStrokeActuatorMain = fMaxStrokeActuatorMain; *)
(* end *)

(* fLengthActuatorKnuckle         = sqrt(fLengthAKnuckle^2 + fLengthBKnuckle^2 -(2*fLengthAKnuckle*fLengthBKnuckle*cosd(fAngleKnuckleArmAct))); *)
(* fStrokeActuatorKnuckle         = fLengthActuatorKnuckle - fMinLengthActuatorKnuckle; *)

(* if fStrokeActuatorKnuckle < 0 *)
(* fStrokeActuatorKnuckle = 0; *)
(* elseif fStrokeActuatorKnuckle > fMaxStrokeActuatorKnuckle *)
(* fMaxStrokeActuatorKnuckle = fMaxStrokeActuatorKnuckle; *)
(* end *)
(* '<S1>:1:71' fHeightMain                 = fHeightPlatformKing + fHeightKingSlew + fHeightSlewTop; *)
(* x = fLengthPlatform*cos(fTheta1) + fHeightMain*cos(fTheta1 + pi/2) + fLengthMainArm*cos(fTheta1 + fTheta3) + fLengthKnuckleArm * cos (fTheta1 + fTheta3 + fTheta4 - pi/2); *)
(* y = fHeightPlatform + fLengthPlatform*sin(fTheta1) + fHeightMain * sin(fTheta1 + pi/2) + fLengthMainArm *sin(fTheta1 + fTheta3) + fLengthKnuckleArm*sin(fTheta1 + fTheta3 + fTheta4 - pi/2); *)
(* '<S1>:1:76' x = fLengthPlatform*cos(fTheta1) + fHeightMain*cos(fTheta1 + pi/2) + fLengthMainArm*cos(fTheta1 + fTheta3) + fLengthKnuckleArm * cos (fTheta1 + fTheta3 + fTheta4 - pi/2); *)
(* '<S1>:1:77' y = fHeightPlatform + fLengthPlatform*sin(fTheta1) + fHeightMain * sin(fTheta1 + pi/2) + fLengthMainArm *sin(fTheta1 + fTheta3) + fLengthKnuckleArm*sin(fTheta1 + fTheta3 + fTheta4 - pi/2); *)
x_tmp := fTheta1 + fTheta3;
x_tmp_0 := (x_tmp + fTheta4) - 1.5707963267948966;
(* Outport: '<Root>/x' incorporates:
 *  MATLAB Function: '<Root>/Forward kinematics actuator strokes' *)
x := (((COS(fTheta1 + 1.5707963267948966) * 1.424) + (1.3 * COS(fTheta1))) + (COS(x_tmp) * 1.5)) + (COS(x_tmp_0) * 1.158);
(* Outport: '<Root>/y' incorporates:
 *  MATLAB Function: '<Root>/Forward kinematics actuator strokes' *)
y := ((((1.3 * SIN(fTheta1)) + 1.402) + (SIN(fTheta1 + 1.5707963267948966) * 1.424)) + (SIN(x_tmp) * 1.5)) + (SIN(x_tmp_0) * 1.158);

END_FUNCTION_BLOCK

// ---- MACHINE CONTROL/KinematicFunctions2d/FB_WireLengthOnCraneFunction.TcPOU
FUNCTION_BLOCK FB_WireLengthOnCraneFunction
VAR_INPUT
	fTheta3: LREAL;
	fTheta4: LREAL;
END_VAR
VAR_OUTPUT
	wireLengthOnCrane: LREAL;
END_VAR
VAR
	Ps1x: LREAL;
	Ps1y: LREAL;
	Ps2x: LREAL;
	Ps2y: LREAL;
	Ps3x: LREAL;
	Ps3y: LREAL;
	b_a: LREAL;
	d_a: LREAL;
	Ps1x_tmp: LREAL;
	Ps1x_tmp_0: LREAL;
	Ps3x_tmp_tmp: LREAL;
END_VAR


(* MATLAB Function: '<Root>/wireLengthOnCraneFunction1' *)
(* MATLAB Function 'wireLengthOnCraneFunction1': '<S1>:1' *)
(* '<S1>:1:3' lengthOrigoToWinch = 0.2199; *)
(* '<S1>:1:4' heightOrigoToWinch = 0.0895; *)
(* '<S1>:1:5' lengthOrigoToSheave1 = 0.2348; *)
(* '<S1>:1:6' heightOrigoToSheave1 = 0.060; *)
(* '<S1>:1:7' lengthOrigoToSheave2 = 1.520; *)
(* '<S1>:1:8' heigthOrigoToSheave2 = 0.095; *)
(* '<S1>:1:9' lengthMainArmToSheave3 = 0.2591; *)
(* '<S1>:1:10' lengthMainArmToSheave4 = 1.158; *)
(* '<S1>:1:11' offsetAngleSheave3deg = 49.7; *)
(* '<S1>:1:12' offsetAngleSheave3rad = deg2rad(offsetAngleSheave3deg); *)
(* '<S1>:1:13' offsetAngleSheave4deg = 90; *)
(* '<S1>:1:14' offsetAngleSheave4rad = deg2rad(offsetAngleSheave4deg); *)
(* '<S1>:1:16' lengthMainArm = 1.500; *)
(* '<S1>:1:17' pitchRadiusWinch = 0.0716; *)
(* '<S1>:1:18' pitchRadiusSheave = 0.034; *)
(* '<S1>:1:20' Pwx = -lengthOrigoToWinch; *)
(* '<S1>:1:21' Pwy = -heightOrigoToWinch; *)
(* '<S1>:1:22' Ps1x = lengthOrigoToSheave1 * cos(theta3) - heightOrigoToSheave1 * sin(theta3); *)
Ps1x_tmp := SIN(fTheta3);
Ps1x_tmp_0 := COS(fTheta3);
Ps1x := (0.2348 * Ps1x_tmp_0) - (0.06 * Ps1x_tmp);
(* '<S1>:1:23' Ps1y = lengthOrigoToSheave1 * sin(theta3) + heightOrigoToSheave1 * cos(theta3); *)
Ps1y := (0.2348 * Ps1x_tmp) + (0.06 * Ps1x_tmp_0);
(* '<S1>:1:24' Ps2x = lengthOrigoToSheave2 * cos(theta3) - heigthOrigoToSheave2 * sin(theta3); *)
Ps2x := (1.52 * Ps1x_tmp_0) - (0.095 * Ps1x_tmp);
(* '<S1>:1:25' Ps2y = lengthOrigoToSheave2 * sin(theta3) + heigthOrigoToSheave2 * cos(theta3); *)
Ps2y := (1.52 * Ps1x_tmp) + (0.095 * Ps1x_tmp_0);
(* '<S1>:1:26' Ps3x = lengthMainArm * cos(theta3) + lengthMainArmToSheave3 * cos(theta3 + theta4 - offsetAngleSheave3rad); *)
Ps3x_tmp_tmp := fTheta3 + fTheta4;
Ps3x := (COS(Ps3x_tmp_tmp - 0.86742863824118188) * 0.2591) + (1.5 * Ps1x_tmp_0);
(* '<S1>:1:27' Ps3y = lengthMainArm * sin(theta3) + lengthMainArmToSheave3 * sin(theta3 + theta4 - offsetAngleSheave3rad); *)
Ps3y := (SIN(Ps3x_tmp_tmp - 0.86742863824118188) * 0.2591) + (1.5 * Ps1x_tmp);
(* '<S1>:1:28' Ps4x = lengthMainArm * cos(theta3) + lengthMainArmToSheave4 * cos(theta3 + theta4 - offsetAngleSheave4rad); *)
(* '<S1>:1:29' Ps4y = lengthMainArm * sin(theta3) + lengthMainArmToSheave4 * sin(theta3 + theta4 - offsetAngleSheave4rad); *)
(* '<S1>:1:31' distanceWinchSheave1 =  sqrt((Ps1x - Pwx)^2 + (Ps1y - Pwy)^2); *)
Ps1x_tmp := SQRT(((Ps1x - -0.2199) * (Ps1x - -0.2199)) + ((Ps1y - -0.0895) * (Ps1y - -0.0895)));
(* distanceTwoPoints(Pwx, Pwy, Ps1x, Ps1y); *)
(* '<S1>:1:32' distanceSheave1Sheave2 = sqrt((Ps2x - Ps1x)^2 + (Ps2y - Ps1y)^2); *)
Ps1x_tmp_0 := Ps2x - Ps1x;
b_a := Ps2y - Ps1y;
Ps1x_tmp_0 := SQRT((Ps1x_tmp_0 * Ps1x_tmp_0) + (b_a * b_a));
(* distanceTwoPoints(Ps2x, Ps2y, Ps1x, Ps1y); *)
(* '<S1>:1:33' distanceSheave2Sheave3 = sqrt((Ps3x - Ps2x)^2 + (Ps3y - Ps2y)^2); *)
b_a := Ps3x - Ps2x;
d_a := Ps3y - Ps2y;
b_a := SQRT((b_a * b_a) + (d_a * d_a));
(* distanceTwoPoints(Ps2x, Ps2y, Ps3x, Ps3y); *)
(* '<S1>:1:34' distanceSheave3Sheave4 = sqrt((Ps4x - Ps3x)^2 + (Ps4y - Ps3y)^2); *)
d_a := ((COS(Ps3x_tmp_tmp - 1.5707963267948966) * 1.158) + (1.5 * COS(fTheta3))) - Ps3x;
Ps3x_tmp_tmp := ((SIN(Ps3x_tmp_tmp - 1.5707963267948966) * 1.158) + (1.5 * SIN(fTheta3))) - Ps3y;
d_a := SQRT((d_a * d_a) + (Ps3x_tmp_tmp * Ps3x_tmp_tmp));
(* Outport: '<Root>/wireLengthOnCrane' incorporates:
 *  MATLAB Function: '<Root>/wireLengthOnCraneFunction1' *)
(* distanceTwoPoints(Ps4x, Ps4y, Ps3x, Ps3y); *)
(* '<S1>:1:36' tangentLengthWinchSheave1 = sqrt(distanceWinchSheave1^2 -(pitchRadiusWinch -pitchRadiusSheave)^2); *)
(* tangentLengthFunction(distanceWinchSheave1, pitchRadiusWinch, pitchRadiusSheave); *)
(* '<S1>:1:37' tangentLengthSheave1Sheave2 = sqrt(distanceSheave1Sheave2^2 -(pitchRadiusSheave -pitchRadiusSheave)^2); *)
(* tangentLengthFunction(distanceSheave1Sheave2, pitchRadiusSheave, pitchRadiusSheave); *)
(* '<S1>:1:38' tangentLengthSheave2Sheave3 = sqrt(distanceSheave2Sheave3^2 -(pitchRadiusSheave -pitchRadiusSheave)^2); *)
(* tangentLengthFunction(distanceSheave2Sheave3, pitchRadiusSheave, pitchRadiusSheave); *)
(* '<S1>:1:39' tangentLengthSheave3Sheave4 = sqrt(distanceSheave3Sheave4^2 -(pitchRadiusSheave -pitchRadiusSheave)^2); *)
(* tangentLengthFunction(distanceSheave3Sheave4, pitchRadiusSheave, pitchRadiusSheave); *)
(* '<S1>:1:41' offsetAngleDeg = 113.6 + 9.9; *)
(* '<S1>:1:42' offsetAngleRad = deg2rad(offsetAngleDeg); *)
(* '<S1>:1:44' wrapAngle = offsetAngleRad - theta3 - theta4; *)
(* '<S1>:1:45' wrapLength = wrapAngle * pitchRadiusSheave; *)
(* '<S1>:1:47' wireLengthOnCrane = tangentLengthWinchSheave1 + tangentLengthSheave1Sheave2 + tangentLengthSheave2Sheave3 + tangentLengthSheave3Sheave4 + wrapLength; *)
wireLengthOnCrane := (((SQRT((Ps1x_tmp * Ps1x_tmp) - 0.0014137599999999996) + SQRT(Ps1x_tmp_0 * Ps1x_tmp_0)) + SQRT(b_a * b_a)) + SQRT(d_a * d_a)) + (((2.155481626212997 - fTheta3) - fTheta4) * 0.034);

END_FUNCTION_BLOCK

// ---- AXIS CONTROL/P_AxisControl.TcPOU
PROGRAM P_AxisControl
VAR
END_VAR

//Axis Control program based on youtube series Twincat 3 NC Videos MB05a until MB17b plus MB22 by @electricalautomation https://www.youtube.com/watch?v=BxRAOdTks9I&list=PL762SfoJC-e8NbAUQ-H7a_TOdqrlBPCw4&index=25

IF G_Inputs.bManualModeSelector THEN
	Manual_mode();
ELSIF G_Inputs.bAutoModeSelector THEN
	Auto_mode();
ELSE
	Stop_mode();
END_IF

METHOD Auto_mode : BOOL
VAR_INPUT
END_VAR
//AXIS 1 Main arm actuator

G_AXIS1.lrBC_PowerOverride := 100;

G_AXIS1.bBC_ResetExe := G_Inputs.bJoystickLeftEnable OR G_Inputs.bGreenButton OR G_AXIS1.bBC_MoveAbsDone;

//Power Enable
G_AXIS1.bBC_PowerEnCmd := G_Inputs.bAutoModeSelector;
G_AXIS1.bBC_PowerEnNegative := G_Inputs.bAutoModeSelector;
G_AXIS1.bBC_PowerEnPositive := G_Inputs.bAutoModeSelector;

G_AXIS1.lrBC_MoveAbsPosition := G_InverseKinematics.fStrokeActuatorMainInverse*1000;
G_AXIS1.lrBC_MoveAbsVelocity := 20;
G_AXIS1.bBC_MoveAbsExe := G_Inputs.bGreenButton;


//Position control
IF G_Inputs.bJoystickLeftEnable AND G_AXIS1.bBC_MoveAbsDone THEN
	G_AXIS1.bBC_ExtSetGenDisExe := FALSE;
	G_AXIS1.bBC_ExtSetGenEnaExe := TRUE;
ELSE
	G_AXIS1.bBC_ExtSetGenDisExe := TRUE;
	G_AXIS1.bBC_ExtSetGenEnaExe := FALSE;
END_IF


G_AXIS1.lrBC_MoveAddPos := G_InverseKinematics.fStrokeActuatorMainInverse*1000;


//Update axis
AXIS1_LD_Auto();


//Axis 3 Knuckle arm actuator

G_AXIS3.lrTC_PowerOverride := 100;

G_AXIS3.bTC_ResetExe := G_Inputs.bJoystickLeftEnable OR G_Inputs.bGreenButton OR G_AXIS3.bTC_MoveAbsDone;

//Power Enable
G_AXIS3.bTC_PowerEnCmd := G_Inputs.bAutoModeSelector;
G_AXIS3.bTC_PowerEnNegative := G_Inputs.bAutoModeSelector;
G_AXIS3.bTC_PowerEnPositive := G_Inputs.bAutoModeSelector;

G_AXIS3.lrTC_MoveAbsPosition := G_InverseKinematics.fStrokeActuatorKnuckleInverse*1000;
G_AXIS3.lrTC_MoveAbsVelocity := 20;
G_AXIS3.bTC_MoveAbsExe := G_Inputs.bGreenButton;


//Position control
IF G_Inputs.bJoystickLeftEnable AND G_AXIS3.bTC_MoveAbsDone THEN
	G_AXIS3.bTC_ExtSetGenDisExe := FALSE;
	G_AXIS3.bTC_ExtSetGenEnaExe := TRUE;
ELSE
	G_AXIS3.bTC_ExtSetGenDisExe := TRUE;
	G_AXIS3.bTC_ExtSetGenEnaExe := FALSE;
END_IF


G_AXIS3.lrTC_MoveAddPos := G_InverseKinematics.fStrokeActuatorKnuckleInverse*1000;


//Update axis
AXIS3_LD_Auto();


//Axis 4 Winch motor

G_AXIS4.lrWM_PowerOverride := 50;

G_AXIS4.bWM_ResetExe := G_Inputs.bGreenButton OR G_AXIS1.bBC_MoveAbsDone;
//GVL_AXIS4.bWM_ResetExe := G_Inputs.bJoystickRightEnable OR G_Inputs.bGreenButton OR GVL_AXIS1.bBC_MoveAbsDone;

//Power Enable
G_AXIS4.bWM_PowerEnCmd := G_Inputs.bAutoModeSelector;
G_AXIS4.bWM_PowerEnNegative := G_Inputs.bAutoModeSelector;
G_AXIS4.bWM_PowerEnPositive := G_Inputs.bAutoModeSelector;

//G_AXIS4.lrWM_MoveAbsPosition := G_MachineControl.fWinchMotorAngleRef*180/PI;
//G_AXIS4.lrWM_MoveAbsVelocity := 50;
//G_AXIS4.bWM_MoveAbsExe := G_Inputs.bGreenButton;

//Position control
IF G_Inputs.bJoystickLeftEnable AND G_AXIS1.bBC_MoveAbsDone AND G_AXIS3.bTC_MoveAbsDone THEN
	G_AXIS4.bWM_ExtSetGenDisExe := FALSE;
	G_AXIS4.bWM_ExtSetGenEnaExe := TRUE;
ELSE
	G_AXIS4.bWM_ExtSetGenDisExe := TRUE;
	G_AXIS4.bWM_ExtSetGenEnaExe := FALSE;
END_IF

G_AXIS4.lrWM_MoveSetPointVel := 500;
G_AXIS4.lrWM_MoveAddPos := G_MachineControl.fWinchMotorAngleAbsRef; //G_MachineControl.fWinchMotorAngleRef*180/PI; //Convert to degrees


//Update axis
AXIS4_LD_Auto();
END_METHOD

METHOD AXIS1_LD_Auto : BOOL
VAR_INPUT
END_VAR
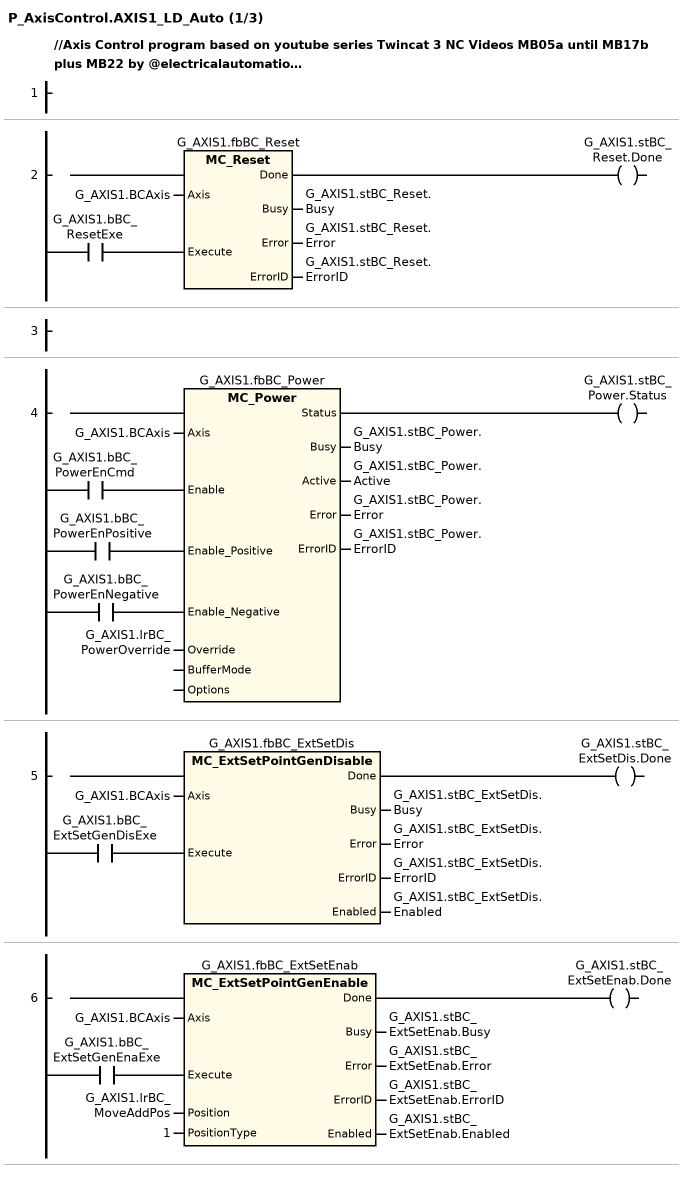
// NETWORK 1: //Axis Control program based on youtube series Twincat 3 NC Videos MB05a until MB17b plus MB22 by @electricalautomation https://www.youtube.com/watch?v=BxRAOdTks9I&list=PL762SfoJC-e8NbAUQ-H7a_TOdqrlBPCw4&index=25

// NETWORK 2
G_AXIS1.fbBC_Reset(
    Axis := G_AXIS1.BCAxis,
    Execute := G_AXIS1.bBC_ResetExe,
    Busy => G_AXIS1.stBC_Reset.Busy,
    Error => G_AXIS1.stBC_Reset.Error,
    ErrorID => G_AXIS1.stBC_Reset.ErrorID); // MC_Reset
G_AXIS1.stBC_Reset.Done := G_AXIS1.fbBC_Reset.Done;

// NETWORK 3

// NETWORK 4
G_AXIS1.fbBC_Power(
    Axis := G_AXIS1.BCAxis,
    Enable := G_AXIS1.bBC_PowerEnCmd,
    Enable_Positive := G_AXIS1.bBC_PowerEnPositive,
    Enable_Negative := G_AXIS1.bBC_PowerEnNegative,
    Override := G_AXIS1.lrBC_PowerOverride,
    Busy => G_AXIS1.stBC_Power.Busy,
    Active => G_AXIS1.stBC_Power.Active,
    Error => G_AXIS1.stBC_Power.Error,
    ErrorID => G_AXIS1.stBC_Power.ErrorID); // MC_Power
G_AXIS1.stBC_Power.Status := G_AXIS1.fbBC_Power.Status;

// NETWORK 5
G_AXIS1.fbBC_ExtSetDis(
    Axis := G_AXIS1.BCAxis,
    Execute := G_AXIS1.bBC_ExtSetGenDisExe,
    Busy => G_AXIS1.stBC_ExtSetDis.Busy,
    Error => G_AXIS1.stBC_ExtSetDis.Error,
    ErrorID => G_AXIS1.stBC_ExtSetDis.ErrorID,
    Enabled => G_AXIS1.stBC_ExtSetDis.Enabled); // MC_ExtSetPointGenDisable
G_AXIS1.stBC_ExtSetDis.Done := G_AXIS1.fbBC_ExtSetDis.Done;

// NETWORK 6
G_AXIS1.fbBC_ExtSetEnab(
    Axis := G_AXIS1.BCAxis,
    Execute := G_AXIS1.bBC_ExtSetGenEnaExe,
    Position := G_AXIS1.lrBC_MoveAddPos,
    PositionType := 1,
    Busy => G_AXIS1.stBC_ExtSetEnab.Busy,
    Error => G_AXIS1.stBC_ExtSetEnab.Error,
    ErrorID => G_AXIS1.stBC_ExtSetEnab.ErrorID,
    Enabled => G_AXIS1.stBC_ExtSetEnab.Enabled); // MC_ExtSetPointGenEnable
G_AXIS1.stBC_ExtSetEnab.Done := G_AXIS1.fbBC_ExtSetEnab.Done;

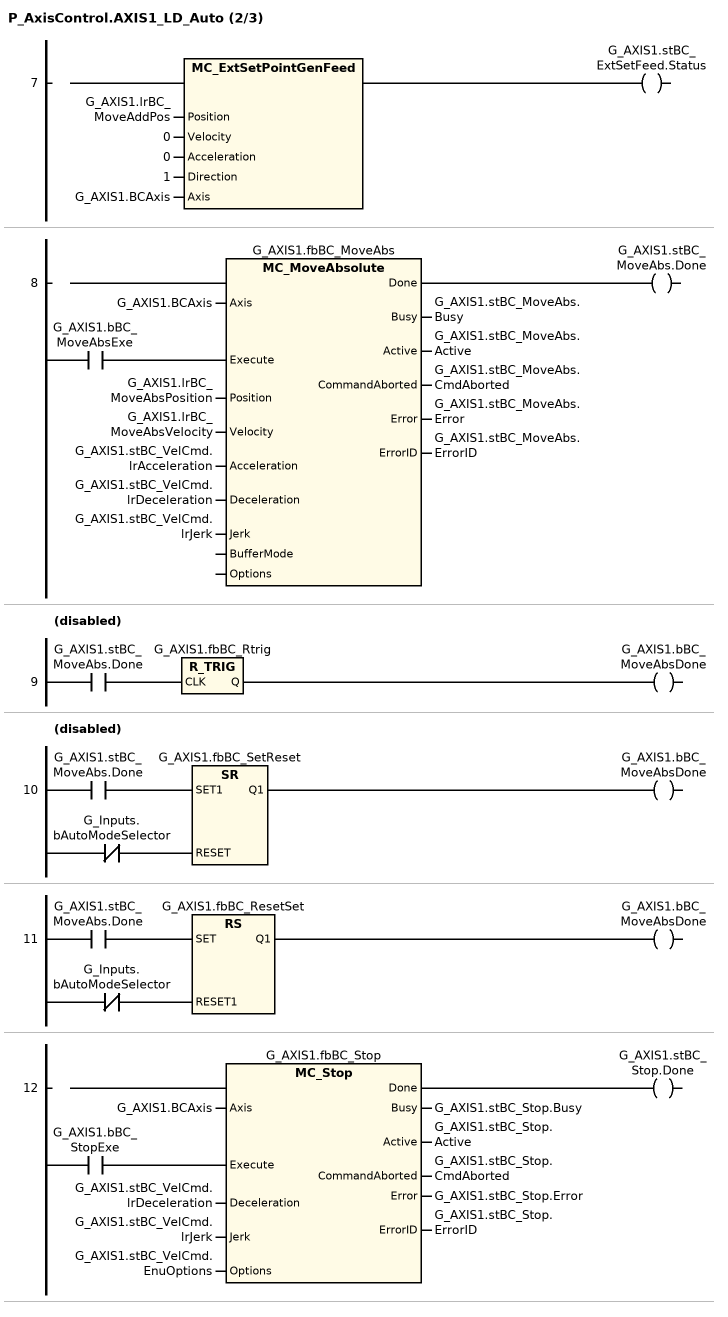
// NETWORK 7
G_AXIS1.stBC_ExtSetFeed.Status := MC_ExtSetPointGenFeed(Position := G_AXIS1.lrBC_MoveAddPos, Velocity := 0, Acceleration := 0, Direction := 1, Axis := G_AXIS1.BCAxis);

// NETWORK 8
G_AXIS1.fbBC_MoveAbs(
    Axis := G_AXIS1.BCAxis,
    Execute := G_AXIS1.bBC_MoveAbsExe,
    Position := G_AXIS1.lrBC_MoveAbsPosition,
    Velocity := G_AXIS1.lrBC_MoveAbsVelocity,
    Acceleration := G_AXIS1.stBC_VelCmd.lrAcceleration,
    Deceleration := G_AXIS1.stBC_VelCmd.lrDeceleration,
    Jerk := G_AXIS1.stBC_VelCmd.lrJerk,
    Busy => G_AXIS1.stBC_MoveAbs.Busy,
    Active => G_AXIS1.stBC_MoveAbs.Active,
    CommandAborted => G_AXIS1.stBC_MoveAbs.CmdAborted,
    Error => G_AXIS1.stBC_MoveAbs.Error,
    ErrorID => G_AXIS1.stBC_MoveAbs.ErrorID); // MC_MoveAbsolute
G_AXIS1.stBC_MoveAbs.Done := G_AXIS1.fbBC_MoveAbs.Done;

// NETWORK 9 (disabled)
// G_AXIS1.fbBC_Rtrig(CLK := G_AXIS1.stBC_MoveAbs.Done); // R_TRIG
// G_AXIS1.bBC_MoveAbsDone := G_AXIS1.fbBC_Rtrig.Q;

// NETWORK 10 (disabled)
// G_AXIS1.fbBC_SetReset(SET1 := G_AXIS1.stBC_MoveAbs.Done, RESET := NOT G_Inputs.bAutoModeSelector); // SR
// G_AXIS1.bBC_MoveAbsDone := G_AXIS1.fbBC_SetReset.Q1;

// NETWORK 11
G_AXIS1.fbBC_ResetSet(SET := G_AXIS1.stBC_MoveAbs.Done, RESET1 := NOT G_Inputs.bAutoModeSelector); // RS
G_AXIS1.bBC_MoveAbsDone := G_AXIS1.fbBC_ResetSet.Q1;

// NETWORK 12
G_AXIS1.fbBC_Stop(
    Axis := G_AXIS1.BCAxis,
    Execute := G_AXIS1.bBC_StopExe,
    Deceleration := G_AXIS1.stBC_VelCmd.lrDeceleration,
    Jerk := G_AXIS1.stBC_VelCmd.lrJerk,
    Options := G_AXIS1.stBC_VelCmd.EnuOptions,
    Busy => G_AXIS1.stBC_Stop.Busy,
    Active => G_AXIS1.stBC_Stop.Active,
    CommandAborted => G_AXIS1.stBC_Stop.CmdAborted,
    Error => G_AXIS1.stBC_Stop.Error,
    ErrorID => G_AXIS1.stBC_Stop.ErrorID); // MC_Stop
G_AXIS1.stBC_Stop.Done := G_AXIS1.fbBC_Stop.Done;

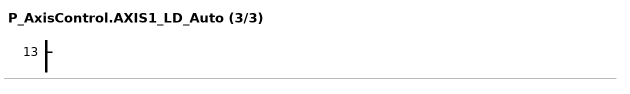
// NETWORK 13
END_METHOD

METHOD AXIS1_LD_Manual : BOOL
VAR_INPUT
END_VAR
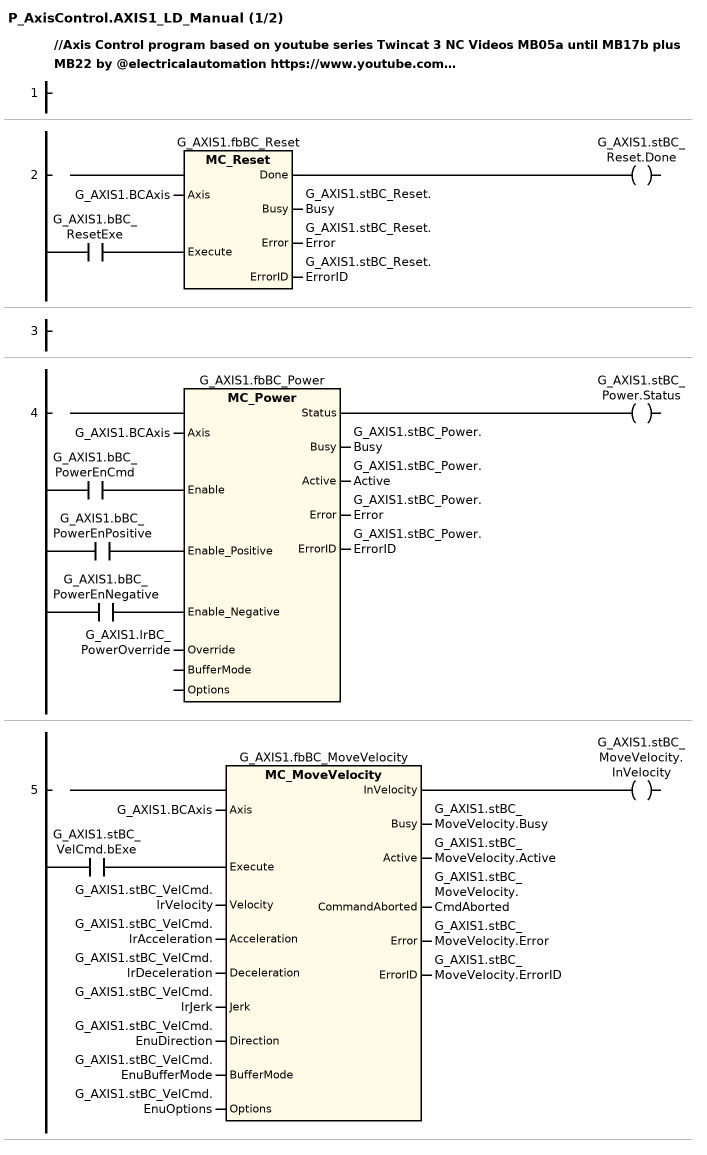
// NETWORK 1: //Axis Control program based on youtube series Twincat 3 NC Videos MB05a until MB17b plus MB22 by @electricalautomation https://www.youtube.com/watch?v=BxRAOdTks9I&list=PL762SfoJC-e8NbAUQ-H7a_TOdqrlBPCw4&index=25

// NETWORK 2
G_AXIS1.fbBC_Reset(
    Axis := G_AXIS1.BCAxis,
    Execute := G_AXIS1.bBC_ResetExe,
    Busy => G_AXIS1.stBC_Reset.Busy,
    Error => G_AXIS1.stBC_Reset.Error,
    ErrorID => G_AXIS1.stBC_Reset.ErrorID); // MC_Reset
G_AXIS1.stBC_Reset.Done := G_AXIS1.fbBC_Reset.Done;

// NETWORK 3

// NETWORK 4
G_AXIS1.fbBC_Power(
    Axis := G_AXIS1.BCAxis,
    Enable := G_AXIS1.bBC_PowerEnCmd,
    Enable_Positive := G_AXIS1.bBC_PowerEnPositive,
    Enable_Negative := G_AXIS1.bBC_PowerEnNegative,
    Override := G_AXIS1.lrBC_PowerOverride,
    Busy => G_AXIS1.stBC_Power.Busy,
    Active => G_AXIS1.stBC_Power.Active,
    Error => G_AXIS1.stBC_Power.Error,
    ErrorID => G_AXIS1.stBC_Power.ErrorID); // MC_Power
G_AXIS1.stBC_Power.Status := G_AXIS1.fbBC_Power.Status;

// NETWORK 5
G_AXIS1.fbBC_MoveVelocity(
    Axis := G_AXIS1.BCAxis,
    Execute := G_AXIS1.stBC_VelCmd.bExe,
    Velocity := G_AXIS1.stBC_VelCmd.lrVelocity,
    Acceleration := G_AXIS1.stBC_VelCmd.lrAcceleration,
    Deceleration := G_AXIS1.stBC_VelCmd.lrDeceleration,
    Jerk := G_AXIS1.stBC_VelCmd.lrJerk,
    Direction := G_AXIS1.stBC_VelCmd.EnuDirection,
    BufferMode := G_AXIS1.stBC_VelCmd.EnuBufferMode,
    Options := G_AXIS1.stBC_VelCmd.EnuOptions,
    Busy => G_AXIS1.stBC_MoveVelocity.Busy,
    Active => G_AXIS1.stBC_MoveVelocity.Active,
    CommandAborted => G_AXIS1.stBC_MoveVelocity.CmdAborted,
    Error => G_AXIS1.stBC_MoveVelocity.Error,
    ErrorID => G_AXIS1.stBC_MoveVelocity.ErrorID); // MC_MoveVelocity
G_AXIS1.stBC_MoveVelocity.InVelocity := G_AXIS1.fbBC_MoveVelocity.InVelocity;

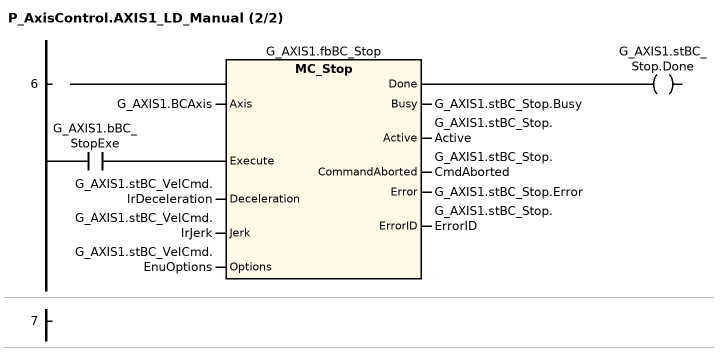
// NETWORK 6
G_AXIS1.fbBC_Stop(
    Axis := G_AXIS1.BCAxis,
    Execute := G_AXIS1.bBC_StopExe,
    Deceleration := G_AXIS1.stBC_VelCmd.lrDeceleration,
    Jerk := G_AXIS1.stBC_VelCmd.lrJerk,
    Options := G_AXIS1.stBC_VelCmd.EnuOptions,
    Busy => G_AXIS1.stBC_Stop.Busy,
    Active => G_AXIS1.stBC_Stop.Active,
    CommandAborted => G_AXIS1.stBC_Stop.CmdAborted,
    Error => G_AXIS1.stBC_Stop.Error,
    ErrorID => G_AXIS1.stBC_Stop.ErrorID); // MC_Stop
G_AXIS1.stBC_Stop.Done := G_AXIS1.fbBC_Stop.Done;

// NETWORK 7
END_METHOD

METHOD AXIS2_LD_Manual : BOOL
VAR_INPUT
END_VAR
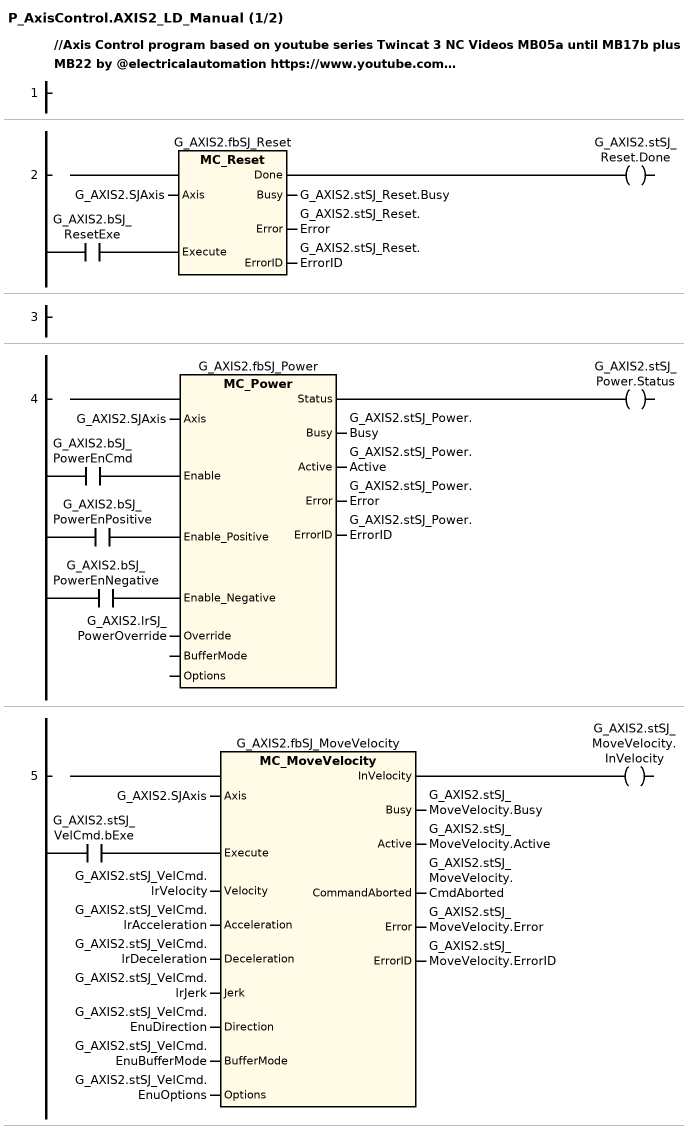
// NETWORK 1: //Axis Control program based on youtube series Twincat 3 NC Videos MB05a until MB17b plus MB22 by @electricalautomation https://www.youtube.com/watch?v=BxRAOdTks9I&list=PL762SfoJC-e8NbAUQ-H7a_TOdqrlBPCw4&index=25

// NETWORK 2
G_AXIS2.fbSJ_Reset(
    Axis := G_AXIS2.SJAxis,
    Execute := G_AXIS2.bSJ_ResetExe,
    Busy => G_AXIS2.stSJ_Reset.Busy,
    Error => G_AXIS2.stSJ_Reset.Error,
    ErrorID => G_AXIS2.stSJ_Reset.ErrorID); // MC_Reset
G_AXIS2.stSJ_Reset.Done := G_AXIS2.fbSJ_Reset.Done;

// NETWORK 3

// NETWORK 4
G_AXIS2.fbSJ_Power(
    Axis := G_AXIS2.SJAxis,
    Enable := G_AXIS2.bSJ_PowerEnCmd,
    Enable_Positive := G_AXIS2.bSJ_PowerEnPositive,
    Enable_Negative := G_AXIS2.bSJ_PowerEnNegative,
    Override := G_AXIS2.lrSJ_PowerOverride,
    Busy => G_AXIS2.stSJ_Power.Busy,
    Active => G_AXIS2.stSJ_Power.Active,
    Error => G_AXIS2.stSJ_Power.Error,
    ErrorID => G_AXIS2.stSJ_Power.ErrorID); // MC_Power
G_AXIS2.stSJ_Power.Status := G_AXIS2.fbSJ_Power.Status;

// NETWORK 5
G_AXIS2.fbSJ_MoveVelocity(
    Axis := G_AXIS2.SJAxis,
    Execute := G_AXIS2.stSJ_VelCmd.bExe,
    Velocity := G_AXIS2.stSJ_VelCmd.lrVelocity,
    Acceleration := G_AXIS2.stSJ_VelCmd.lrAcceleration,
    Deceleration := G_AXIS2.stSJ_VelCmd.lrDeceleration,
    Jerk := G_AXIS2.stSJ_VelCmd.lrJerk,
    Direction := G_AXIS2.stSJ_VelCmd.EnuDirection,
    BufferMode := G_AXIS2.stSJ_VelCmd.EnuBufferMode,
    Options := G_AXIS2.stSJ_VelCmd.EnuOptions,
    Busy => G_AXIS2.stSJ_MoveVelocity.Busy,
    Active => G_AXIS2.stSJ_MoveVelocity.Active,
    CommandAborted => G_AXIS2.stSJ_MoveVelocity.CmdAborted,
    Error => G_AXIS2.stSJ_MoveVelocity.Error,
    ErrorID => G_AXIS2.stSJ_MoveVelocity.ErrorID); // MC_MoveVelocity
G_AXIS2.stSJ_MoveVelocity.InVelocity := G_AXIS2.fbSJ_MoveVelocity.InVelocity;

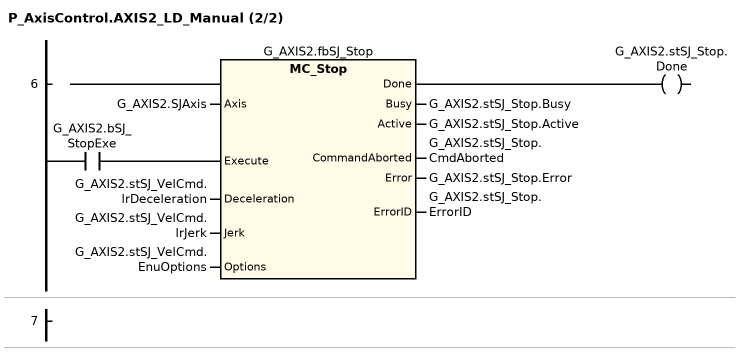
// NETWORK 6
G_AXIS2.fbSJ_Stop(
    Axis := G_AXIS2.SJAxis,
    Execute := G_AXIS2.bSJ_StopExe,
    Deceleration := G_AXIS2.stSJ_VelCmd.lrDeceleration,
    Jerk := G_AXIS2.stSJ_VelCmd.lrJerk,
    Options := G_AXIS2.stSJ_VelCmd.EnuOptions,
    Busy => G_AXIS2.stSJ_Stop.Busy,
    Active => G_AXIS2.stSJ_Stop.Active,
    CommandAborted => G_AXIS2.stSJ_Stop.CmdAborted,
    Error => G_AXIS2.stSJ_Stop.Error,
    ErrorID => G_AXIS2.stSJ_Stop.ErrorID); // MC_Stop
G_AXIS2.stSJ_Stop.Done := G_AXIS2.fbSJ_Stop.Done;

// NETWORK 7
END_METHOD

METHOD AXIS3_LD_Auto : BOOL
VAR_INPUT
END_VAR
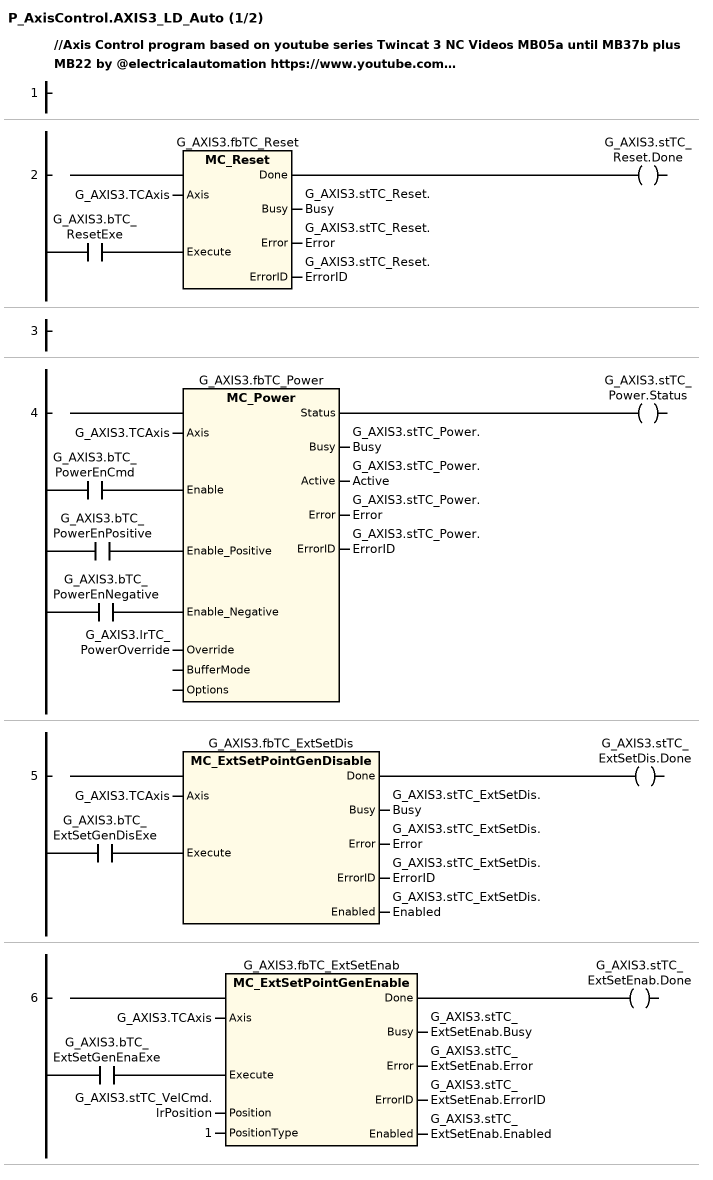
// NETWORK 1: //Axis Control program based on youtube series Twincat 3 NC Videos MB05a until MB37b plus MB22 by @electricalautomation https://www.youtube.com/watch?v=BxRAOdTks9I&list=PL762SfoJC-e8NbAUQ-H7a_TOdqrlBPCw4&index=25

// NETWORK 2
G_AXIS3.fbTC_Reset(
    Axis := G_AXIS3.TCAxis,
    Execute := G_AXIS3.bTC_ResetExe,
    Busy => G_AXIS3.stTC_Reset.Busy,
    Error => G_AXIS3.stTC_Reset.Error,
    ErrorID => G_AXIS3.stTC_Reset.ErrorID); // MC_Reset
G_AXIS3.stTC_Reset.Done := G_AXIS3.fbTC_Reset.Done;

// NETWORK 3

// NETWORK 4
G_AXIS3.fbTC_Power(
    Axis := G_AXIS3.TCAxis,
    Enable := G_AXIS3.bTC_PowerEnCmd,
    Enable_Positive := G_AXIS3.bTC_PowerEnPositive,
    Enable_Negative := G_AXIS3.bTC_PowerEnNegative,
    Override := G_AXIS3.lrTC_PowerOverride,
    Busy => G_AXIS3.stTC_Power.Busy,
    Active => G_AXIS3.stTC_Power.Active,
    Error => G_AXIS3.stTC_Power.Error,
    ErrorID => G_AXIS3.stTC_Power.ErrorID); // MC_Power
G_AXIS3.stTC_Power.Status := G_AXIS3.fbTC_Power.Status;

// NETWORK 5
G_AXIS3.fbTC_ExtSetDis(
    Axis := G_AXIS3.TCAxis,
    Execute := G_AXIS3.bTC_ExtSetGenDisExe,
    Busy => G_AXIS3.stTC_ExtSetDis.Busy,
    Error => G_AXIS3.stTC_ExtSetDis.Error,
    ErrorID => G_AXIS3.stTC_ExtSetDis.ErrorID,
    Enabled => G_AXIS3.stTC_ExtSetDis.Enabled); // MC_ExtSetPointGenDisable
G_AXIS3.stTC_ExtSetDis.Done := G_AXIS3.fbTC_ExtSetDis.Done;

// NETWORK 6
G_AXIS3.fbTC_ExtSetEnab(
    Axis := G_AXIS3.TCAxis,
    Execute := G_AXIS3.bTC_ExtSetGenEnaExe,
    Position := G_AXIS3.stTC_VelCmd.lrPosition,
    PositionType := 1,
    Busy => G_AXIS3.stTC_ExtSetEnab.Busy,
    Error => G_AXIS3.stTC_ExtSetEnab.Error,
    ErrorID => G_AXIS3.stTC_ExtSetEnab.ErrorID,
    Enabled => G_AXIS3.stTC_ExtSetEnab.Enabled); // MC_ExtSetPointGenEnable
G_AXIS3.stTC_ExtSetEnab.Done := G_AXIS3.fbTC_ExtSetEnab.Done;

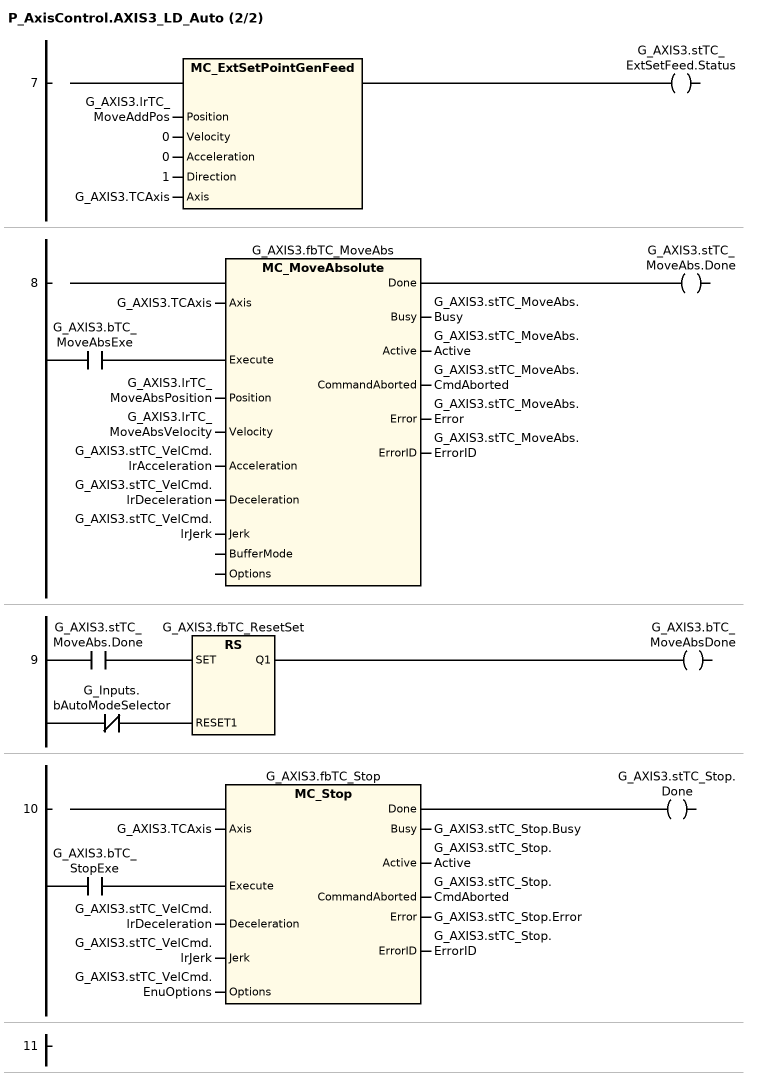
// NETWORK 7
G_AXIS3.stTC_ExtSetFeed.Status := MC_ExtSetPointGenFeed(Position := G_AXIS3.lrTC_MoveAddPos, Velocity := 0, Acceleration := 0, Direction := 1, Axis := G_AXIS3.TCAxis);

// NETWORK 8
G_AXIS3.fbTC_MoveAbs(
    Axis := G_AXIS3.TCAxis,
    Execute := G_AXIS3.bTC_MoveAbsExe,
    Position := G_AXIS3.lrTC_MoveAbsPosition,
    Velocity := G_AXIS3.lrTC_MoveAbsVelocity,
    Acceleration := G_AXIS3.stTC_VelCmd.lrAcceleration,
    Deceleration := G_AXIS3.stTC_VelCmd.lrDeceleration,
    Jerk := G_AXIS3.stTC_VelCmd.lrJerk,
    Busy => G_AXIS3.stTC_MoveAbs.Busy,
    Active => G_AXIS3.stTC_MoveAbs.Active,
    CommandAborted => G_AXIS3.stTC_MoveAbs.CmdAborted,
    Error => G_AXIS3.stTC_MoveAbs.Error,
    ErrorID => G_AXIS3.stTC_MoveAbs.ErrorID); // MC_MoveAbsolute
G_AXIS3.stTC_MoveAbs.Done := G_AXIS3.fbTC_MoveAbs.Done;

// NETWORK 9
G_AXIS3.fbTC_ResetSet(SET := G_AXIS3.stTC_MoveAbs.Done, RESET1 := NOT G_Inputs.bAutoModeSelector); // RS
G_AXIS3.bTC_MoveAbsDone := G_AXIS3.fbTC_ResetSet.Q1;

// NETWORK 10
G_AXIS3.fbTC_Stop(
    Axis := G_AXIS3.TCAxis,
    Execute := G_AXIS3.bTC_StopExe,
    Deceleration := G_AXIS3.stTC_VelCmd.lrDeceleration,
    Jerk := G_AXIS3.stTC_VelCmd.lrJerk,
    Options := G_AXIS3.stTC_VelCmd.EnuOptions,
    Busy => G_AXIS3.stTC_Stop.Busy,
    Active => G_AXIS3.stTC_Stop.Active,
    CommandAborted => G_AXIS3.stTC_Stop.CmdAborted,
    Error => G_AXIS3.stTC_Stop.Error,
    ErrorID => G_AXIS3.stTC_Stop.ErrorID); // MC_Stop
G_AXIS3.stTC_Stop.Done := G_AXIS3.fbTC_Stop.Done;

// NETWORK 11
END_METHOD

METHOD AXIS3_LD_Manual : BOOL
VAR_INPUT
END_VAR
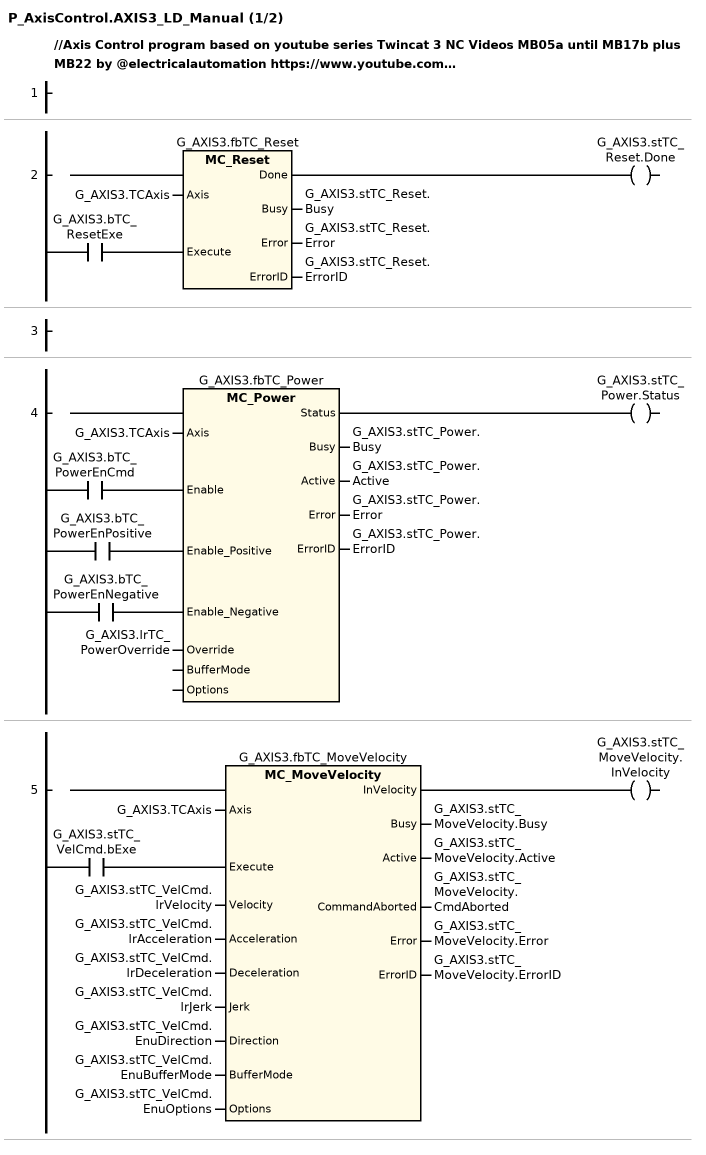
// NETWORK 1: //Axis Control program based on youtube series Twincat 3 NC Videos MB05a until MB17b plus MB22 by @electricalautomation https://www.youtube.com/watch?v=BxRAOdTks9I&list=PL762SfoJC-e8NbAUQ-H7a_TOdqrlBPCw4&index=25

// NETWORK 2
G_AXIS3.fbTC_Reset(
    Axis := G_AXIS3.TCAxis,
    Execute := G_AXIS3.bTC_ResetExe,
    Busy => G_AXIS3.stTC_Reset.Busy,
    Error => G_AXIS3.stTC_Reset.Error,
    ErrorID => G_AXIS3.stTC_Reset.ErrorID); // MC_Reset
G_AXIS3.stTC_Reset.Done := G_AXIS3.fbTC_Reset.Done;

// NETWORK 3

// NETWORK 4
G_AXIS3.fbTC_Power(
    Axis := G_AXIS3.TCAxis,
    Enable := G_AXIS3.bTC_PowerEnCmd,
    Enable_Positive := G_AXIS3.bTC_PowerEnPositive,
    Enable_Negative := G_AXIS3.bTC_PowerEnNegative,
    Override := G_AXIS3.lrTC_PowerOverride,
    Busy => G_AXIS3.stTC_Power.Busy,
    Active => G_AXIS3.stTC_Power.Active,
    Error => G_AXIS3.stTC_Power.Error,
    ErrorID => G_AXIS3.stTC_Power.ErrorID); // MC_Power
G_AXIS3.stTC_Power.Status := G_AXIS3.fbTC_Power.Status;

// NETWORK 5
G_AXIS3.fbTC_MoveVelocity(
    Axis := G_AXIS3.TCAxis,
    Execute := G_AXIS3.stTC_VelCmd.bExe,
    Velocity := G_AXIS3.stTC_VelCmd.lrVelocity,
    Acceleration := G_AXIS3.stTC_VelCmd.lrAcceleration,
    Deceleration := G_AXIS3.stTC_VelCmd.lrDeceleration,
    Jerk := G_AXIS3.stTC_VelCmd.lrJerk,
    Direction := G_AXIS3.stTC_VelCmd.EnuDirection,
    BufferMode := G_AXIS3.stTC_VelCmd.EnuBufferMode,
    Options := G_AXIS3.stTC_VelCmd.EnuOptions,
    Busy => G_AXIS3.stTC_MoveVelocity.Busy,
    Active => G_AXIS3.stTC_MoveVelocity.Active,
    CommandAborted => G_AXIS3.stTC_MoveVelocity.CmdAborted,
    Error => G_AXIS3.stTC_MoveVelocity.Error,
    ErrorID => G_AXIS3.stTC_MoveVelocity.ErrorID); // MC_MoveVelocity
G_AXIS3.stTC_MoveVelocity.InVelocity := G_AXIS3.fbTC_MoveVelocity.InVelocity;

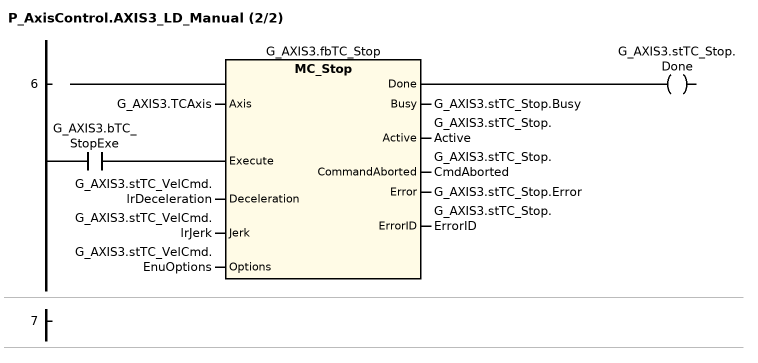
// NETWORK 6
G_AXIS3.fbTC_Stop(
    Axis := G_AXIS3.TCAxis,
    Execute := G_AXIS3.bTC_StopExe,
    Deceleration := G_AXIS3.stTC_VelCmd.lrDeceleration,
    Jerk := G_AXIS3.stTC_VelCmd.lrJerk,
    Options := G_AXIS3.stTC_VelCmd.EnuOptions,
    Busy => G_AXIS3.stTC_Stop.Busy,
    Active => G_AXIS3.stTC_Stop.Active,
    CommandAborted => G_AXIS3.stTC_Stop.CmdAborted,
    Error => G_AXIS3.stTC_Stop.Error,
    ErrorID => G_AXIS3.stTC_Stop.ErrorID); // MC_Stop
G_AXIS3.stTC_Stop.Done := G_AXIS3.fbTC_Stop.Done;

// NETWORK 7
END_METHOD

METHOD AXIS4_LD_Auto : BOOL
VAR_INPUT
END_VAR
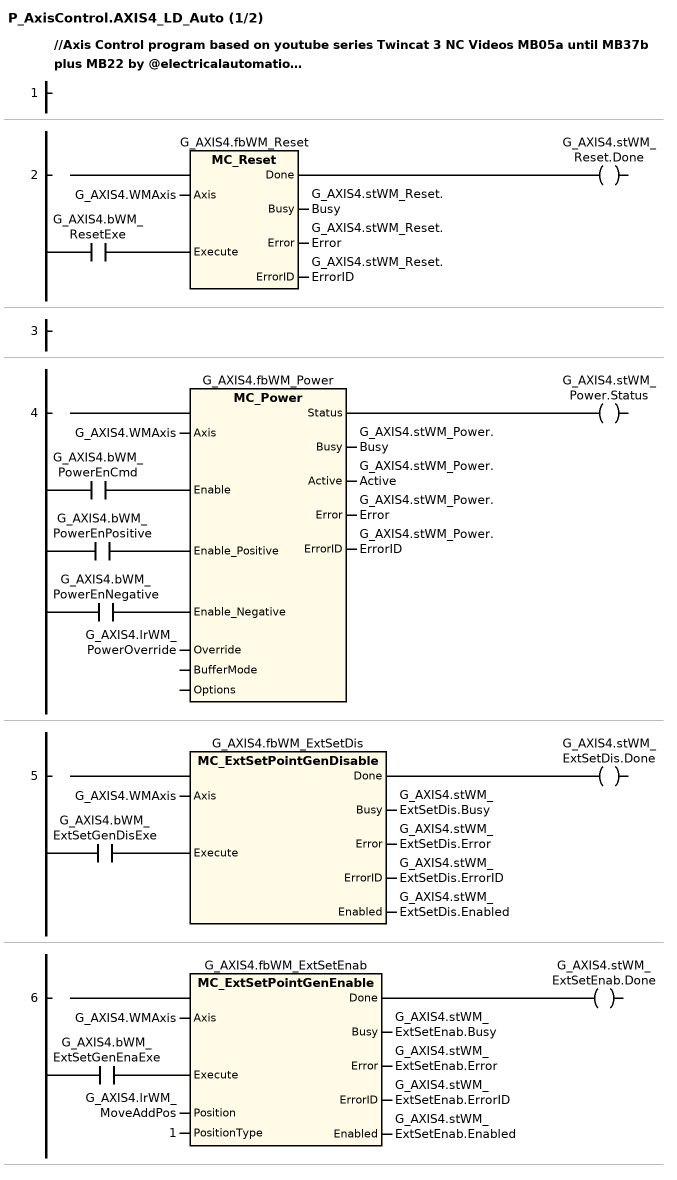
// NETWORK 1: //Axis Control program based on youtube series Twincat 3 NC Videos MB05a until MB37b plus MB22 by @electricalautomation https://www.youtube.com/waWMh?v=BxRAOdTks9I&list=PL762SfoJC-e8NbAUQ-H7a_TOdqrlBPCw4&index=25

// NETWORK 2
G_AXIS4.fbWM_Reset(
    Axis := G_AXIS4.WMAxis,
    Execute := G_AXIS4.bWM_ResetExe,
    Busy => G_AXIS4.stWM_Reset.Busy,
    Error => G_AXIS4.stWM_Reset.Error,
    ErrorID => G_AXIS4.stWM_Reset.ErrorID); // MC_Reset
G_AXIS4.stWM_Reset.Done := G_AXIS4.fbWM_Reset.Done;

// NETWORK 3

// NETWORK 4
G_AXIS4.fbWM_Power(
    Axis := G_AXIS4.WMAxis,
    Enable := G_AXIS4.bWM_PowerEnCmd,
    Enable_Positive := G_AXIS4.bWM_PowerEnPositive,
    Enable_Negative := G_AXIS4.bWM_PowerEnNegative,
    Override := G_AXIS4.lrWM_PowerOverride,
    Busy => G_AXIS4.stWM_Power.Busy,
    Active => G_AXIS4.stWM_Power.Active,
    Error => G_AXIS4.stWM_Power.Error,
    ErrorID => G_AXIS4.stWM_Power.ErrorID); // MC_Power
G_AXIS4.stWM_Power.Status := G_AXIS4.fbWM_Power.Status;

// NETWORK 5
G_AXIS4.fbWM_ExtSetDis(
    Axis := G_AXIS4.WMAxis,
    Execute := G_AXIS4.bWM_ExtSetGenDisExe,
    Busy => G_AXIS4.stWM_ExtSetDis.Busy,
    Error => G_AXIS4.stWM_ExtSetDis.Error,
    ErrorID => G_AXIS4.stWM_ExtSetDis.ErrorID,
    Enabled => G_AXIS4.stWM_ExtSetDis.Enabled); // MC_ExtSetPointGenDisable
G_AXIS4.stWM_ExtSetDis.Done := G_AXIS4.fbWM_ExtSetDis.Done;

// NETWORK 6
G_AXIS4.fbWM_ExtSetEnab(
    Axis := G_AXIS4.WMAxis,
    Execute := G_AXIS4.bWM_ExtSetGenEnaExe,
    Position := G_AXIS4.lrWM_MoveAddPos,
    PositionType := 1,
    Busy => G_AXIS4.stWM_ExtSetEnab.Busy,
    Error => G_AXIS4.stWM_ExtSetEnab.Error,
    ErrorID => G_AXIS4.stWM_ExtSetEnab.ErrorID,
    Enabled => G_AXIS4.stWM_ExtSetEnab.Enabled); // MC_ExtSetPointGenEnable
G_AXIS4.stWM_ExtSetEnab.Done := G_AXIS4.fbWM_ExtSetEnab.Done;

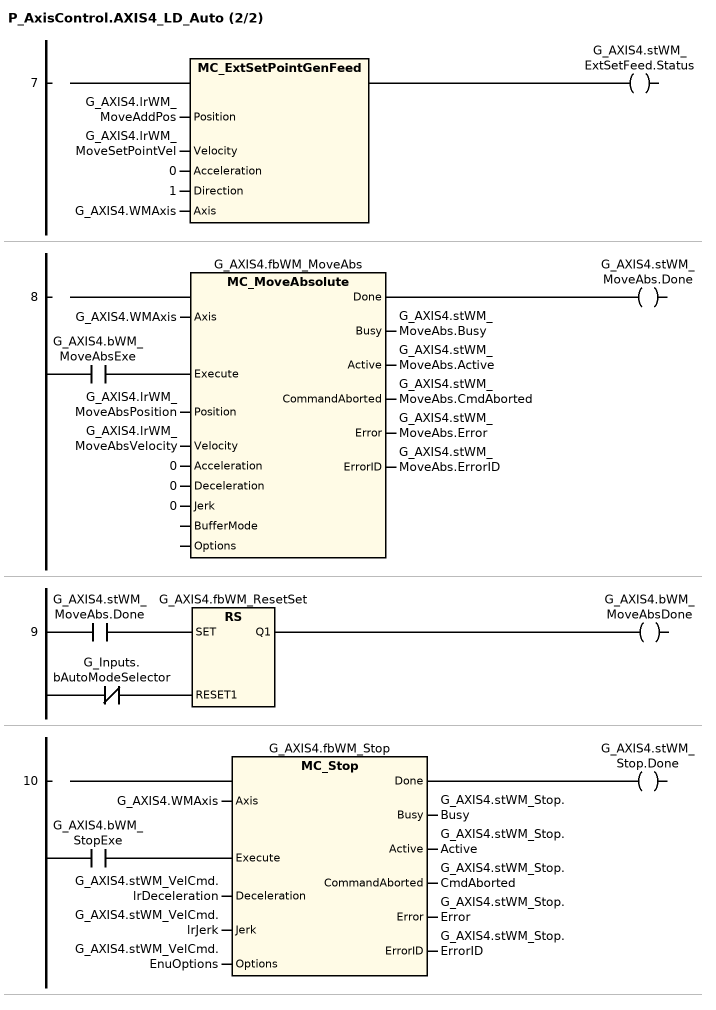
// NETWORK 7
G_AXIS4.stWM_ExtSetFeed.Status := MC_ExtSetPointGenFeed(Position := G_AXIS4.lrWM_MoveAddPos, Velocity := G_AXIS4.lrWM_MoveSetPointVel, Acceleration := 0, Direction := 1, Axis := G_AXIS4.WMAxis);

// NETWORK 8
G_AXIS4.fbWM_MoveAbs(
    Axis := G_AXIS4.WMAxis,
    Execute := G_AXIS4.bWM_MoveAbsExe,
    Position := G_AXIS4.lrWM_MoveAbsPosition,
    Velocity := G_AXIS4.lrWM_MoveAbsVelocity,
    Acceleration := 0,
    Deceleration := 0,
    Jerk := 0,
    Busy => G_AXIS4.stWM_MoveAbs.Busy,
    Active => G_AXIS4.stWM_MoveAbs.Active,
    CommandAborted => G_AXIS4.stWM_MoveAbs.CmdAborted,
    Error => G_AXIS4.stWM_MoveAbs.Error,
    ErrorID => G_AXIS4.stWM_MoveAbs.ErrorID); // MC_MoveAbsolute
G_AXIS4.stWM_MoveAbs.Done := G_AXIS4.fbWM_MoveAbs.Done;

// NETWORK 9
G_AXIS4.fbWM_ResetSet(SET := G_AXIS4.stWM_MoveAbs.Done, RESET1 := NOT G_Inputs.bAutoModeSelector); // RS
G_AXIS4.bWM_MoveAbsDone := G_AXIS4.fbWM_ResetSet.Q1;

// NETWORK 10
G_AXIS4.fbWM_Stop(
    Axis := G_AXIS4.WMAxis,
    Execute := G_AXIS4.bWM_StopExe,
    Deceleration := G_AXIS4.stWM_VelCmd.lrDeceleration,
    Jerk := G_AXIS4.stWM_VelCmd.lrJerk,
    Options := G_AXIS4.stWM_VelCmd.EnuOptions,
    Busy => G_AXIS4.stWM_Stop.Busy,
    Active => G_AXIS4.stWM_Stop.Active,
    CommandAborted => G_AXIS4.stWM_Stop.CmdAborted,
    Error => G_AXIS4.stWM_Stop.Error,
    ErrorID => G_AXIS4.stWM_Stop.ErrorID); // MC_Stop
G_AXIS4.stWM_Stop.Done := G_AXIS4.fbWM_Stop.Done;
END_METHOD

METHOD AXIS4_LD_Manual : BOOL
VAR_INPUT
END_VAR
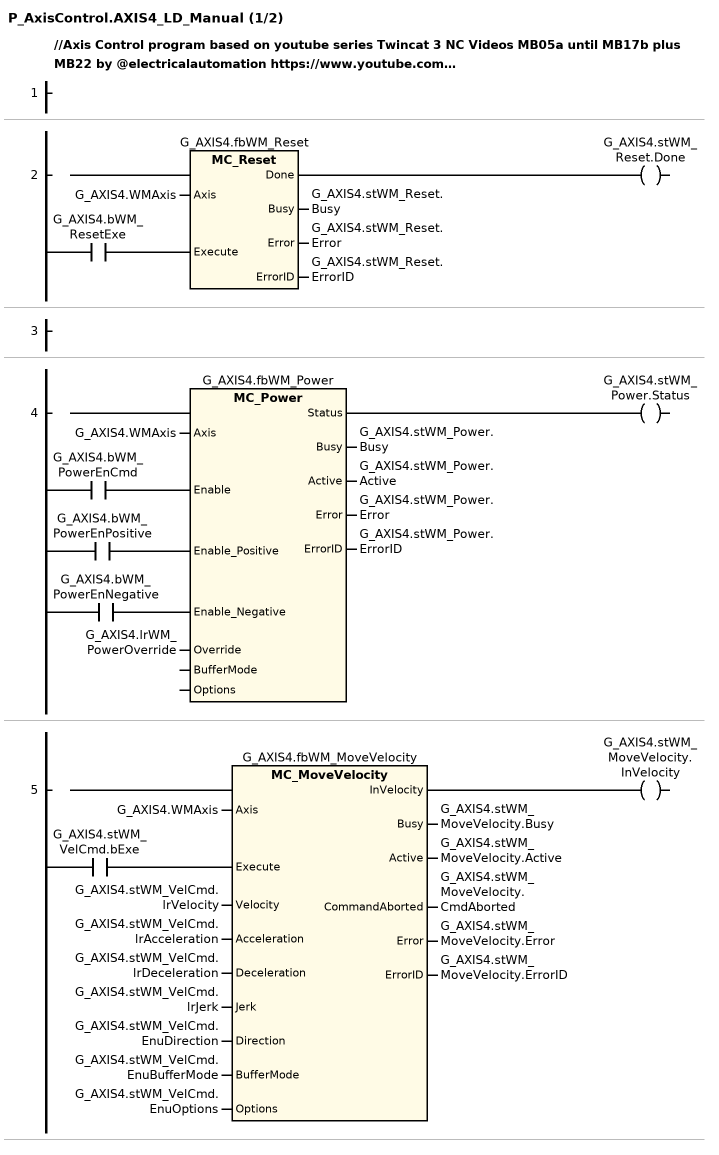
// NETWORK 1: //Axis Control program based on youtube series Twincat 3 NC Videos MB05a until MB17b plus MB22 by @electricalautomation https://www.youtube.com/watch?v=BxRAOdTks9I&list=PL762SfoJC-e8NbAUQ-H7a_TOdqrlBPCw4&index=25

// NETWORK 2
G_AXIS4.fbWM_Reset(
    Axis := G_AXIS4.WMAxis,
    Execute := G_AXIS4.bWM_ResetExe,
    Busy => G_AXIS4.stWM_Reset.Busy,
    Error => G_AXIS4.stWM_Reset.Error,
    ErrorID => G_AXIS4.stWM_Reset.ErrorID); // MC_Reset
G_AXIS4.stWM_Reset.Done := G_AXIS4.fbWM_Reset.Done;

// NETWORK 3

// NETWORK 4
G_AXIS4.fbWM_Power(
    Axis := G_AXIS4.WMAxis,
    Enable := G_AXIS4.bWM_PowerEnCmd,
    Enable_Positive := G_AXIS4.bWM_PowerEnPositive,
    Enable_Negative := G_AXIS4.bWM_PowerEnNegative,
    Override := G_AXIS4.lrWM_PowerOverride,
    Busy => G_AXIS4.stWM_Power.Busy,
    Active => G_AXIS4.stWM_Power.Active,
    Error => G_AXIS4.stWM_Power.Error,
    ErrorID => G_AXIS4.stWM_Power.ErrorID); // MC_Power
G_AXIS4.stWM_Power.Status := G_AXIS4.fbWM_Power.Status;

// NETWORK 5
G_AXIS4.fbWM_MoveVelocity(
    Axis := G_AXIS4.WMAxis,
    Execute := G_AXIS4.stWM_VelCmd.bExe,
    Velocity := G_AXIS4.stWM_VelCmd.lrVelocity,
    Acceleration := G_AXIS4.stWM_VelCmd.lrAcceleration,
    Deceleration := G_AXIS4.stWM_VelCmd.lrDeceleration,
    Jerk := G_AXIS4.stWM_VelCmd.lrJerk,
    Direction := G_AXIS4.stWM_VelCmd.EnuDirection,
    BufferMode := G_AXIS4.stWM_VelCmd.EnuBufferMode,
    Options := G_AXIS4.stWM_VelCmd.EnuOptions,
    Busy => G_AXIS4.stWM_MoveVelocity.Busy,
    Active => G_AXIS4.stWM_MoveVelocity.Active,
    CommandAborted => G_AXIS4.stWM_MoveVelocity.CmdAborted,
    Error => G_AXIS4.stWM_MoveVelocity.Error,
    ErrorID => G_AXIS4.stWM_MoveVelocity.ErrorID); // MC_MoveVelocity
G_AXIS4.stWM_MoveVelocity.InVelocity := G_AXIS4.fbWM_MoveVelocity.InVelocity;

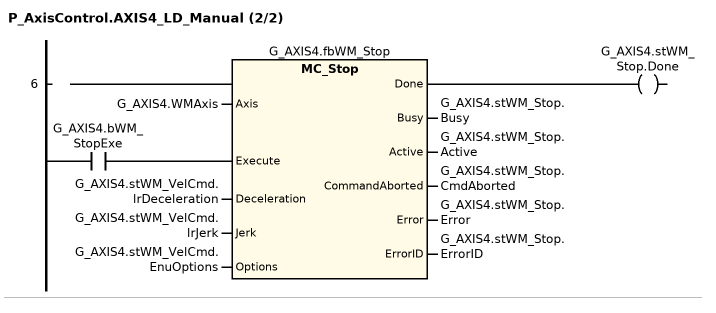
// NETWORK 6
G_AXIS4.fbWM_Stop(
    Axis := G_AXIS4.WMAxis,
    Execute := G_AXIS4.bWM_StopExe,
    Deceleration := G_AXIS4.stWM_VelCmd.lrDeceleration,
    Jerk := G_AXIS4.stWM_VelCmd.lrJerk,
    Options := G_AXIS4.stWM_VelCmd.EnuOptions,
    Busy => G_AXIS4.stWM_Stop.Busy,
    Active => G_AXIS4.stWM_Stop.Active,
    CommandAborted => G_AXIS4.stWM_Stop.CmdAborted,
    Error => G_AXIS4.stWM_Stop.Error,
    ErrorID => G_AXIS4.stWM_Stop.ErrorID); // MC_Stop
G_AXIS4.stWM_Stop.Done := G_AXIS4.fbWM_Stop.Done;
END_METHOD

METHOD Manual_mode : BOOL
VAR_INPUT
END_VAR
//Axis 1 Main arm actuator
AXIS1_LD_Manual();

G_AXIS1.bBC_ResetExe := FALSE;

G_AXIS1.stBC_VelCmd.EnuDirection := MC_Undefined_Direction;

G_AXIS1.stBC_VelCmd.bExe := FALSE;

G_AXIS1.bBC_PowerEnCmd := G_Inputs.bManualModeSelector;

IF G_Sensors.fJoystickLeftNormalizedX  > 0 AND G_Inputs.bJoystickLeftEnable THEN
	G_AXIS1.bBC_PowerEnNegative := TRUE;
	G_AXIS1.stBC_VelCmd.EnuDirection := MC_Negative_Direction;
	G_AXIS1.lrBC_PowerOverride := ABS(G_Sensors.fJoystickLeftNormalizedX) * 100;	
	G_AXIS1.stBC_VelCmd.bExe := TRUE;
ELSIF G_Sensors.fJoystickLeftNormalizedX < 0 AND G_Inputs.bJoystickLeftEnable THEN
	G_AXIS1.bBC_PowerEnPositive := TRUE;
	G_AXIS1.stBC_VelCmd.EnuDirection := MC_Positive_Direction;
	G_AXIS1.lrBC_PowerOverride := ABS(G_Sensors.fJoystickLeftNormalizedX) * 100;	
	G_AXIS1.stBC_VelCmd.bExe := TRUE;
ELSE
	 G_AXIS1.lrBC_PowerOverride := 0;
	 G_AXIS1.stBC_VelCmd.bExe := FALSE;
	 G_AXIS1.bBC_PowerEnNegative := FALSE;
	 G_AXIS1.bBC_PowerEnPositive := FALSE;
END_IF

G_AXIS1.bBC_ResetExe := TRUE;


//Axis 2 Slew joint actuator
AXIS2_LD_Manual();

G_AXIS2.bSJ_ResetExe := FALSE;

G_AXIS2.stSJ_VelCmd.EnuDirection := MC_Undefined_Direction;

G_AXIS2.stSJ_VelCmd.bExe := FALSE;

G_AXIS2.bSJ_PowerEnCmd := G_Inputs.bManualModeSelector;

IF G_Sensors.fJoystickRightNormalizedX  > 0 AND G_Inputs.bJoystickRightEnable THEN
	G_AXIS2.bSJ_PowerEnPositive := TRUE;
	G_AXIS2.stSJ_VelCmd.EnuDirection := MC_Positive_Direction;
	G_AXIS2.lrSJ_PowerOverride := ABS(G_Sensors.fJoystickRightNormalizedX) * 100;	
	G_AXIS2.stSJ_VelCmd.bExe := TRUE;
ELSIF G_Sensors.fJoystickRightNormalizedX < 0 AND G_Inputs.bJoystickRightEnable THEN
	G_AXIS2.bSJ_PowerEnNegative := TRUE;
	G_AXIS2.stSJ_VelCmd.EnuDirection := MC_Negative_Direction;
	G_AXIS2.lrSJ_PowerOverride := ABS(G_Sensors.fJoystickRightNormalizedX) * 100;	
	G_AXIS2.stSJ_VelCmd.bExe := TRUE;
ELSE
	 G_AXIS2.lrSJ_PowerOverride := 0;
	 G_AXIS2.stSJ_VelCmd.bExe := FALSE;
	 G_AXIS2.bSJ_PowerEnNegative := FALSE;
	 G_AXIS2.bSJ_PowerEnPositive := FALSE;
END_IF

G_AXIS2.bSJ_ResetExe := TRUE;


//Axis 3 Knuckle arm actuator
AXIS3_LD_Manual();

G_AXIS3.bTC_ResetExe := FALSE;

G_AXIS3.stTC_VelCmd.EnuDirection := MC_Undefined_Direction;

G_AXIS3.stTC_VelCmd.bExe := FALSE;

G_AXIS3.bTC_PowerEnCmd := G_Inputs.bManualModeSelector;

IF G_Sensors.fJoystickLeftNormalizedY  > 0 AND G_Inputs.bJoystickLeftEnable THEN
	G_AXIS3.bTC_PowerEnPositive := TRUE;
	G_AXIS3.stTC_VelCmd.EnuDirection := MC_Positive_Direction;
	G_AXIS3.lrTC_PowerOverride := ABS(G_Sensors.fJoystickLeftNormalizedY) * 100;	
	G_AXIS3.stTC_VelCmd.bExe := TRUE;
ELSIF G_Sensors.fJoystickLeftNormalizedY < 0 AND G_Inputs.bJoystickLeftEnable THEN
	G_AXIS3.bTC_PowerEnNegative := TRUE;
	G_AXIS3.stTC_VelCmd.EnuDirection := MC_Negative_Direction;
	G_AXIS3.lrTC_PowerOverride := ABS(G_Sensors.fJoystickLeftNormalizedY) * 100;	
	G_AXIS3.stTC_VelCmd.bExe := TRUE;
ELSE
	 G_AXIS3.lrTC_PowerOverride := 0;
	 G_AXIS3.stTC_VelCmd.bExe := FALSE;
	 G_AXIS3.bTC_PowerEnNegative := FALSE;
	 G_AXIS3.bTC_PowerEnPositive := FALSE;
END_IF

G_AXIS3.bTC_ResetExe := TRUE;

(*
AXIS3_LD();

GVL_AXIS3.bTC_ResetExe := G_Inputs.bJoystickLeftEnable;

GVL_AXIS3.EnuMoveVelDirection := G_Sensors.MCDirectionAxis3;

GVL_AXIS3.bTC_PowerEnCmd := G_Inputs.bManualModeSelector;
GVL_AXIS3.bTC_PowerEnNegative := G_Inputs.bManualModeSelector;
GVL_AXIS3.bTC_PowerEnPositive := G_Inputs.bManualModeSelector;


// Velocity control
IF G_Sensors.fJoystickLeftNormalizedY  > 0.01 AND G_Inputs.bJoystickLeftEnable THEN
	GVL_AXIS3.stTC_VelCmd.EnuDirection := MC_Positive_Direction;
	GVL_AXIS3.lrTC_PowerOverride := ABS(G_Sensors.fJoystickLeftNormalizedY) * 100;	
	GVL_AXIS3.stTC_VelCmd.bExe := TRUE;
ELSIF G_Sensors.fJoystickLeftNormalizedY < 0.01 AND G_Inputs.bJoystickLeftEnable THEN
	GVL_AXIS3.stTC_VelCmd.EnuDirection := MC_Negative_Direction;
	GVL_AXIS3.lrTC_PowerOverride := ABS(G_Sensors.fJoystickLeftNormalizedY) * 100;	
	GVL_AXIS3.stTC_VelCmd.bExe := TRUE;
ELSE
	 GVL_AXIS3.lrTC_PowerOverride := 0;
	 //GVL_AXIS3.stTC_VelCmd.EnuDirection := MC_Current_Direction;
	 GVL_AXIS3.stTC_VelCmd.bExe := FALSE;
END_IF
*)

(*
AXIS4_LD();

GVL_AXIS4.bWM_ResetExe := G_Inputs.bJoystickRightEnable;

GVL_AXIS4.EnuMoveVelDirection := G_Sensors.MCDirectionAxis4;

GVL_AXIS4.bWM_PowerEnCmd := G_Inputs.bManualModeSelector;
GVL_AXIS4.bWM_PowerEnNegative := G_Inputs.bManualModeSelector;
GVL_AXIS4.bWM_PowerEnPositive := G_Inputs.bManualModeSelector;


// Velocity control
IF G_Sensors.fJoystickLeftNormalizedY  > 0 AND G_Inputs.bJoystickRightEnable THEN
	GVL_AXIS4.lrWM_PowerOverride := ABS(G_Sensors.fJoystickRightNormalizedY) * 100;
	GVL_AXIS4.stWM_VelCmd.EnuDirection := MC_Positive_Direction;
	GVL_AXIS4.stWM_VelCmd.bExe := TRUE;
ELSIF G_Sensors.fJoystickLeftNormalizedY < 0 AND G_Inputs.bJoystickLeftEnable THEN
	GVL_AXIS4.lrWM_PowerOverride := ABS(G_Sensors.fJoystickLeftNormalizedY) * 100;
	GVL_AXIS4.stWM_VelCmd.EnuDirection := MC_Negative_Direction;
	GVL_AXIS4.stWM_VelCmd.bExe := TRUE;
ELSE
	 GVL_AXIS4.lrWM_PowerOverride := 0;
	 GVL_AXIS4.stWM_VelCmd.EnuDirection := MC_Current_Direction;
	 GVL_AXIS4.stWM_VelCmd.bExe := FALSE;
END_IF
*)

//Axis 4 Winch motor actuator
AXIS4_LD_Manual();

G_AXIS4.bWM_ResetExe := FALSE;

G_AXIS4.stWM_VelCmd.EnuDirection := MC_Undefined_Direction;

G_AXIS4.stWM_VelCmd.bExe := FALSE;

G_AXIS4.bWM_PowerEnCmd := G_Inputs.bManualModeSelector;

IF G_Sensors.fJoystickRightNormalizedY  > 0 AND G_Inputs.bJoystickRightEnable THEN
	G_AXIS4.bWM_PowerEnNegative := TRUE;
	G_AXIS4.stWM_VelCmd.EnuDirection := MC_Negative_Direction;
	G_AXIS4.lrWM_PowerOverride := ABS(G_Sensors.fJoystickRightNormalizedY) * 100;	
	G_AXIS4.stWM_VelCmd.bExe := TRUE;
ELSIF G_Sensors.fJoystickRightNormalizedY < 0 AND G_Inputs.bJoystickRightEnable THEN
	G_AXIS4.bWM_PowerEnPositive := TRUE;
	G_AXIS4.stWM_VelCmd.EnuDirection := MC_Positive_Direction;
	G_AXIS4.lrWM_PowerOverride := ABS(G_Sensors.fJoystickRightNormalizedY) * 100;	
	G_AXIS4.stWM_VelCmd.bExe := TRUE;
ELSE
	 G_AXIS4.lrWM_PowerOverride := 0;
	 G_AXIS4.stWM_VelCmd.bExe := FALSE;
	 G_AXIS4.bWM_PowerEnNegative := FALSE;
	 G_AXIS4.bWM_PowerEnPositive := FALSE;
END_IF

G_AXIS4.bWM_ResetExe := TRUE;
END_METHOD

METHOD Stop_mode : BOOL
VAR_INPUT
END_VAR
//Stop mode

	G_AXIS1.lrBC_PowerOverride := 0;
	G_AXIS1.bBC_StopExe := TRUE;
	G_AXIS1.bBC_PowerEnCmd := FALSE;
	
	AXIS1_LD_Auto();
	AXIS1_LD_Manual();
	
	G_AXIS2.lrSJ_PowerOverride := 0;	
	G_AXIS2.bSJ_StopExe := TRUE;	
	G_AXIS2.bSJ_PowerEnCmd := FALSE;
	
	//AXIS2_LD_Auto();
	AXIS2_LD_Manual();
	
	G_AXIS3.lrTC_PowerOverride := 0;	
	G_AXIS3.bTC_StopExe := TRUE;
	G_AXIS3.bTC_PowerEnCmd := FALSE;
	
	AXIS3_LD_Auto();
	AXIS3_LD_Manual();
	
	G_AXIS4.lrWM_PowerOverride := 0;
	G_AXIS4.bWM_StopExe := TRUE;
	G_AXIS4.bWM_PowerEnCmd := FALSE;
	
	AXIS4_LD_Auto();
	AXIS4_LD_Manual();
END_METHOD

END_PROGRAM

// ---- StablePlatform/P_StablePlatform.TcPOU
PROGRAM P_StablePlatform
VAR
	fbpA 		: FB_AnalogInputScaling;
	fbpB 		: FB_AnalogInputScaling;
	fbpS 	 	: FB_AnalogInputScaling;
	fSVFeedback : FB_AnalogInputScaling;
	fbPistonPos	: FB_AnalogInputScaling_1;
	fbPistonVel	: FB_AnalogInputScaling_1;
	fbJoystick  : FB_JoystickInputScaling;
	fbSVOutput 	: FB_ValveOutput;
	fbAutoModeControl : FB_AutoModeControl; 
	fbLowPassFilter		: FB_LowpassFilter;
END_VAR

// Enable
IF G_StablePlatformIO.bEnable AND G_StablePlatformIO.bEMG_OK THEN
	G_StablePlatformIO.bActivated := TRUE;
ELSE	
	G_StablePlatformIO.bActivated := FALSE;
END_IF
// Mode
IF G_StablePlatformIO.bActivated AND G_StablePlatformIO.bModeSelector AND  G_Inputs.bAutoModeSelector THEN
	G_StablePlatformIO.bAutoMode := TRUE;
	G_StablePlatformIO.bManualMode := FALSE;
	G_StablePlatformIO.fControlSignal :=  G_StablePlatformIO.fAutoModeControlSignal;
ELSIF G_StablePlatformIO.bActivated AND NOT(G_StablePlatformIO.bModeSelector) AND G_Inputs.bManualModeSelector THEN
	G_StablePlatformIO.bAutoMode := FALSE;
	G_StablePlatformIO.bManualMode := TRUE; 
	G_StablePlatformIO.fControlSignal := -G_StablePlatformScaledIO.fJoystickNormalizedX; 	
ELSE
	G_StablePlatformIO.bAutoMode := FALSE;
	G_StablePlatformIO.bManualMode := FALSE; 
	G_StablePlatformIO.fControlSignal := 0.0;
END_IF

// Inputs
fbpA(
	nRawInput := G_StablePlatformIO.npA,
	stAnalogInputScaling := G_StablePlatformParameters.stPressureSensorScaling400bar,
	fOutput => G_StablePlatformScaledIO.bpA
);

fbpB(
	nRawInput := G_StablePlatformIO.npB,
	stAnalogInputScaling := G_StablePlatformParameters.stPressureSensorScaling400bar,
	fOutput => G_StablePlatformScaledIO.bpB
);

fbpS(
	nRawInput := G_StablePlatformIO.npS,
	stAnalogInputScaling := G_StablePlatformParameters.stPressureSensorScaling400bar,
	fOutput => G_StablePlatformScaledIO.bpS
);

fSVFeedback(
	nRawInput := G_StablePlatformIO.nSVFeedback,
	stAnalogInputScaling := G_StablePlatformParameters.stSVFeedbackScaling,
	fOutput => G_StablePlatformScaledIO.fSVFeedback
);

G_StablePlatformScaledIO.fPlatformAngleDeg := F_rad2deg(G_StablePlatformScaledIO.fPlatformAngle);

// Manual Control

fbJoystick(
	bEnable := G_StablePlatformIO.bManualMode,
	nRawInput := G_Inputs.stJoyLX.nValue,
	stJoystickInputScaling := G_StablePlatformParameters.stJoystickInputScalingX,
	fNormalizedOutput => G_StablePlatformScaledIO.fJoystickNormalizedX
);

// Automode Control
fbAutoModeControl(
	bEnable := G_StablePlatformIO.bAutoMode,
	bModeSelector := G_StablePlatformIO.bMotionModeSelector,
	fSampleTime := G_MachineControl.fSampleTime,
	fPistonPosition := G_StablePlatformScaledIO.fPistionPosFiltered,
	fControlSignal => G_StablePlatformIO.fAutoModeControlSignal
);



// Outputs
fbSVOutput(
	bEnable := NOT(G_Inputs.bRedButton) AND G_StablePlatformIO.bActivated,
	bDeadBandCompOn := FALSE,
	stValveDeadBand := G_StablePlatformParameters.stSVValveDeadBand,
	fNormalizedInput := G_StablePlatformIO.fControlSignal,
	nOutput => G_StablePlatformIO.nSVControlSignal
);

G_StablePlatformIO.bSVEnable := G_StablePlatformIO.bActivated;

fbPistonPos(
	nRawInput := G_StablePlatformIO.nPistonPosition,
	stAnalogInputScaling := G_StablePlatformParameters.stPistonPos,
	fOutput => G_StablePlatformScaledIO.fPistonPosition
);

fbLowPassFilter(
	fInput := G_StablePlatformScaledIO.fPistonPosition,
	fDeltaT := G_MachineControl.fSampleTime,
	fCutoffFreq := G_StablePlatformParameters.fCutoffFreq,
	fDamping := G_StablePlatformParameters.fDamping,
	fOutput => G_StablePlatformScaledIO.fPistionPosFiltered
);

fbPistonVel(
	nRawInput := G_StablePlatformIO.nPistonVelocity,
	stAnalogInputScaling := G_StablePlatformParameters.stPistonVel,
	fOutput => G_StablePlatformScaledIO.fPistonVelocity
);


G_StablePlatformScaledIO.fPlatformAngle := fPlatformAngleTheta1(fStroke:=G_StablePlatformScaledIO.fPistionPosFiltered) + F_deg2rad(G_StablePlatformParameters.fAngleOffsetDeg);

END_PROGRAM

// ---- StablePlatform/Function Blocks/FB_AnalogInputScaling_1.TcPOU
FUNCTION_BLOCK FB_AnalogInputScaling_1
VAR_INPUT
	nRawInput 				: INT;
	stAnalogInputScaling    : ST_AnalogInputScaling;
END_VAR
VAR_OUTPUT
	fOutput 				: LREAL;
END_VAR
VAR
	fRawInput 				: LREAL;
	fNormalizedInput		: LREAL;
END_VAR

fRawInput := INT_TO_LREAL(nRawInput);

fNormalizedInput := (fRawInput - stAnalogInputScaling.fMinInputValue) / (stAnalogInputScaling.fMaxInputValue - stAnalogInputScaling.fMinInputValue);

fOutput := LIMIT(stAnalogInputScaling.fMinOutputValue, stAnalogInputScaling.fMinOutputValue + fNormalizedInput*(stAnalogInputScaling.fMaxOutputValue - stAnalogInputScaling.fMinOutputValue), stAnalogInputScaling.fMaxOutputValue);

END_FUNCTION_BLOCK

// ---- StablePlatform/Function Blocks/FB_AutoModeControl.TcPOU
FUNCTION_BLOCK FB_AutoModeControl
VAR_INPUT
	bEnable : BOOL; 
	bModeSelector : BOOL; 
	fSampleTime : LREAL; 
	fPistonPosition : LREAL;
END_VAR
VAR_OUTPUT
	fControlSignal : LREAL;
END_VAR
VAR
	fbCylinderMotionCtonrol : FB_CylinderMotionControl;
	fbClock : FB_Clock;	
	fbRampMotionGenerator : FB_RampMotionGenerator;
	fbWaveMotionGenerator : FB_WaveMotionGenerator;
	bEnableRampMotionGenerator : BOOL;
	bEnableWaveMotionGenerator : BOOL; 
	bRampMotionPlatformCylPos0_m : LREAL; 
	bRampMotionPlatformPositionSP_m : LREAL;

END_VAR

// Enable Motion Mode
IF bEnable AND G_StablePlatformIO.bMotionModeSelector THEN 
	bEnableWaveMotionGenerator := TRUE;
	bEnableRampMotionGenerator := FALSE;
ELSIF bEnable AND NOT(G_StablePlatformIO.bMotionModeSelector) THEN 	
	bEnableWaveMotionGenerator := FALSE;
	bEnableRampMotionGenerator := TRUE;
ELSE
	bEnableWaveMotionGenerator := FALSE;
	bEnableRampMotionGenerator := FALSE;
END_IF

fbClock(
	bEnable := bEnable,
	bStart := G_StablePlatformIO.bStartMotionGenerator,
	bStop := NOT(G_Inputs.bAutoModeSelector OR G_Inputs.bManualModeSelector),
	fCycleTime := fSampleTime,
	fTime => G_StablePlatformIO.fTime
);

// Ramp Motion Generator
bRampMotionPlatformCylPos0_m := F_PlatformAnglePos2CylPos(F_deg2rad(G_StablePlatformIO.bRampMotionPos0_deg));
bRampMotionPlatformPositionSP_m := F_PlatformAnglePos2CylPos(F_deg2rad(G_StablePlatformIO.bRampMotionPositionSP_deg));

fbRampMotionGenerator(
	bEnable := bEnableRampMotionGenerator, 
	bFullPeriode := G_StablePlatformIO.bRampMotionFullPeriode,
	fCylPos0_m := bRampMotionPlatformCylPos0_m,
	fCylVel0_ms := G_StablePlatformIO.bRampMotionCylVel0_ms,
	fPositionSP_m := bRampMotionPlatformPositionSP_m,
	fVelocitySP_ms := G_StablePlatformIO.bRampMotionVelocitySP_ms,
	ft0_s := G_StablePlatformIO.bRampMotiont0_s,
	ftRamp_s := G_StablePlatformIO.bRampMotiontRamp_s,
	ftHoldPos_s := G_StablePlatformIO.bRampMotiontHoldPos_s,
	fSimulationTime_s := fbClock.fTime
);


// Wave Motion Generator
fbWaveMotionGenerator(
	bEnable := bEnableWaveMotionGenerator,
	fBias_deg := 0.0,
	fTheta0_deg := G_StablePlatformIO.fWaveMotionAplitudeTheta0_deg,
	fFreq_rads := G_StablePlatformIO.WaveMotionFreq_rads,
	Fphase_rad := 0.0,
	fCyclicTime_s := fbClock.fTime
);

G_StablePlatformIO.fWaveMotionOmega_degs := fbWaveMotionGenerator.fOmega_degs;
G_StablePlatformIO.fWaveMotionTheta_deg := fbWaveMotionGenerator.fTheta_deg;

IF bEnableRampMotionGenerator THEN
	G_StablePlatformIO.fCylVelRef_ms := fbRampMotionGenerator.VelocityRef_ms;
	G_StablePlatformIO.fCylPosRef_m := fbRampMotionGenerator.PositionRef_m; 
ELSIF bEnableWaveMotionGenerator THEN
	G_StablePlatformIO.fCylVelRef_ms := F_PlatformAngleVel2CylVel(F_deg2rad(G_StablePlatformIO.fWaveMotionTheta_deg),F_deg2rad(G_StablePlatformIO.fWaveMotionOmega_degs));
	G_StablePlatformIO.fCylPosRef_m := F_PlatformAnglePos2CylPos(F_deg2rad(G_StablePlatformIO.fWaveMotionTheta_deg));
ELSE
	G_StablePlatformIO.fCylVelRef_ms := 0.0;
	G_StablePlatformIO.fCylPosRef_m := 0.0;
END_IF

fbCylinderMotionCtonrol(
	ssMethodType :=  BOOL_TO_SINT(bEnable),
	bEnableFeedForward  := G_StablePlatformIO.bEnableFeedForward,
	fMaxValveFlow_lmin := G_StablePlatformIO.fMaxValveFlow_lmin,
	bEnableFeedBackControl := G_StablePlatformIO.bEnableFeedBackControl,
	bEnableIntegralControl := G_StablePlatformIO.bEnableIntegralControl,
	fProportionalGain := G_StablePlatformIO.fProportionalGain,
	fIntegralGain := G_StablePlatformIO.fIntegralGain,
	fMaxPosError_mm := G_StablePlatformIO.fMaxPosError_mm,
	fCylVelRef_ms := G_StablePlatformIO.fCylVelRef_ms,
	fCylPosRef_m := G_StablePlatformIO.fCylPosRef_m,
	fCylPos_m := fPistonPosition
);

IF fbClock.fTime > 0 THEN
	fControlSignal := LIMIT(-G_StablePlatformParameters.fMaxControlSignal, fbCylinderMotionCtonrol.fSvSignal, G_StablePlatformParameters.fMaxControlSignal);
ELSE
	fControlSignal := 0.0;	
END_IF

END_FUNCTION_BLOCK

// ---- StablePlatform/Function Blocks/FB_CylinderMotionControl.TcPOU
FUNCTION_BLOCK FB_CylinderMotionControl
VAR_INPUT
	ssMethodType: SINT;
	bEnableFeedForward: BOOL;
	fMaxValveFlow_lmin: LREAL;
	bEnableFeedBackControl: BOOL;
	bEnableIntegralControl: BOOL;
	fProportionalGain: LREAL;
	fIntegralGain: LREAL;
	fMaxPosError_mm: LREAL;
	fCylVelRef_ms: LREAL;
	fCylPosRef_m: LREAL;
	fCylPos_m: LREAL;
END_VAR
VAR_OUTPUT
	fSvSignal: LREAL;
	fCylPosError_mm: LREAL;
END_VAR
VAR
	rtb_Switch1: LREAL;
	rtb_Reset: LREAL;
	rtb_u_FB: LREAL;
	rtb_Saturation1: LREAL;
	rtb_w_ref: LREAL;
	c_DiscreteTimeIntegrator_DS: LREAL;
	Delay_DSTATE: ARRAY[0..1] OF LREAL;
END_VAR



CASE ssMethodType OF
    0: 
        (* SystemInitialize for Atomic SubSystem: '<Root>/CylinderMotionControl' *)
        (* InitializeConditions for Delay: '<S1>/Delay' *)
        Delay_DSTATE[0] := 0.0;
        Delay_DSTATE[1] := 0.0;
        (* SystemInitialize for Atomic SubSystem: '<S1>/FB_ClosedLoopControl' *)
        (* InitializeConditions for DiscreteIntegrator: '<S2>/Discrete-Time Integrator' *)
        c_DiscreteTimeIntegrator_DS := 0.0;
        (* End of SystemInitialize for SubSystem: '<S1>/FB_ClosedLoopControl' *)
        (* End of SystemInitialize for SubSystem: '<Root>/CylinderMotionControl' *)
    1: 
        (* Outputs for Atomic SubSystem: '<Root>/CylinderMotionControl' *)
        (* Outputs for Atomic SubSystem: '<S1>/FB_OpenLoopControl' *)
        (* Switch: '<S3>/Switch1' incorporates:
         *  Constant: '<S3>/Constant'
         *  Gain: '<S3>/Gain1'
         *  Product: '<S3>/Divide2' *)

        IF bEnableFeedForward THEN 
            (* Switch: '<S3>/Switch2' incorporates:
             *  Constant: '<S3>/Annnulus_Area'
             *  Constant: '<S3>/Bore_Area'
             *  Product: '<S3>/Product1'
             *  Product: '<S3>/Product3' *)

            IF fCylVelRef_ms >= 0.0 THEN 
                rtb_Switch1 := 0.003117 * fCylVelRef_ms;
            ELSE 
                rtb_Switch1 := fCylVelRef_ms * 0.002099;
            END_IF;

            (* End of Switch: '<S3>/Switch2' *)
            rtb_Switch1 := (60000.0 * rtb_Switch1) / fMaxValveFlow_lmin;
        ELSE 
            rtb_Switch1 := 0.0;
        END_IF;

        (* End of Switch: '<S3>/Switch1' *)
        (* End of Outputs for SubSystem: '<S1>/FB_OpenLoopControl' *)
        

        (* Outputs for Atomic SubSystem: '<S1>/FB_ResetIntegralController' *)
        (* MATLAB Function: '<S4>/ResetIntegralController' *)
        (* MATLAB Function 'CylinderMotionControl/FB_ResetIntegralController/ResetIntegralController': '<S5>:1' *)
        (* '<S5>:1:3' if abs(vRef) > 0 || abs(exCyl) > exCylMax *)

        IF ABS(fCylVelRef_ms) > 0.0 THEN 
            ;
            ;
        ELSIF ABS(Delay_DSTATE[0]) > (0.001 * fMaxPosError_mm) THEN 
            ;
            ;
        ELSE 
            (* Outputs for Atomic SubSystem: '<S1>/FB_ClosedLoopControl' *)
            (* DiscreteIntegrator: '<S2>/Discrete-Time Integrator' *)
            (* '<S5>:1:5' else *)
            (* '<S5>:1:6' Reset = 1; *)
            c_DiscreteTimeIntegrator_DS := 0.0;
            (* End of Outputs for SubSystem: '<S1>/FB_ClosedLoopControl' *)
        END_IF;

        (* End of MATLAB Function: '<S4>/ResetIntegralController' *)
        (* End of Outputs for SubSystem: '<S1>/FB_ResetIntegralController' *)
        

        (* Outputs for Atomic SubSystem: '<S1>/FB_ClosedLoopControl' *)
        (* DiscreteIntegrator: '<S2>/Discrete-Time Integrator' *)

        IF c_DiscreteTimeIntegrator_DS >= 1.0 THEN 
            c_DiscreteTimeIntegrator_DS := 1.0;
        ELSIF c_DiscreteTimeIntegrator_DS <= -1.0 THEN 
            c_DiscreteTimeIntegrator_DS := -1.0;
        END_IF;

        (* Sum: '<S2>/Sum1' *)
        rtb_Reset := fCylPosRef_m - fCylPos_m;
        (* Switch: '<S2>/Switch' incorporates:
         *  Constant: '<S2>/Constant'
         *  DiscreteIntegrator: '<S2>/Discrete-Time Integrator' *)

        IF bEnableIntegralControl THEN 
            rtb_u_FB := c_DiscreteTimeIntegrator_DS;
        ELSE 
            rtb_u_FB := 0.0;
        END_IF;

        (* End of Switch: '<S2>/Switch' *)
        

        (* Sum: '<S2>/Sum5' incorporates:
         *  Product: '<S2>/Product' *)
        rtb_u_FB := (fProportionalGain * rtb_Reset) + rtb_u_FB;
        (* Saturate: '<S2>/Saturation1' *)

        IF rtb_u_FB > 1.0 THEN 
            rtb_Saturation1 := 1.0;
        ELSIF rtb_u_FB >= -1.0 THEN 
            rtb_Saturation1 := rtb_u_FB;
        ELSE 
            rtb_Saturation1 := -1.0;
        END_IF;

        (* End of Saturate: '<S2>/Saturation1' *)
        

        (* Switch: '<S2>/Switch1' incorporates:
         *  Constant: '<S2>/Constant1' *)

        IF bEnableFeedBackControl THEN 
            rtb_w_ref := rtb_Saturation1;
        ELSE 
            rtb_w_ref := 0.0;
        END_IF;

        (* End of Switch: '<S2>/Switch1' *)
        

        (* Update for DiscreteIntegrator: '<S2>/Discrete-Time Integrator' incorporates:
         *  Product: '<S2>/Divide'
         *  Product: '<S2>/Product2'
         *  Sum: '<S2>/Sum2'
         *  Sum: '<S2>/Sum3' *)
        c_DiscreteTimeIntegrator_DS := (((((rtb_Saturation1 - rtb_u_FB) / fProportionalGain) + rtb_Reset) * fIntegralGain) * 0.002) + c_DiscreteTimeIntegrator_DS;

        IF c_DiscreteTimeIntegrator_DS >= 1.0 THEN 
            c_DiscreteTimeIntegrator_DS := 1.0;
        ELSIF c_DiscreteTimeIntegrator_DS <= -1.0 THEN 
            c_DiscreteTimeIntegrator_DS := -1.0;
        END_IF;

        (* End of Update for DiscreteIntegrator: '<S2>/Discrete-Time Integrator' *)
        (* End of Outputs for SubSystem: '<S1>/FB_ClosedLoopControl' *)
        

        (* Sum: '<S1>/Add' *)
        fSvSignal := rtb_Switch1 + rtb_w_ref;
        (* Saturate: '<S1>/Saturation' *)

        IF fSvSignal > 1.0 THEN 
            (* Outport: '<Root>/fSvSignal' *)
            fSvSignal := 1.0;
        ELSIF fSvSignal < -1.0 THEN 
            (* Outport: '<Root>/fSvSignal' *)
            fSvSignal := -1.0;
        END_IF;

        (* End of Saturate: '<S1>/Saturation' *)
        

        (* Update for Delay: '<S1>/Delay' *)
        Delay_DSTATE[0] := Delay_DSTATE[1];
        Delay_DSTATE[1] := rtb_Reset;
        (* Outport: '<Root>/fCylPosError_mm' incorporates:
         *  Gain: '<S1>/Gain' *)
        fCylPosError_mm := 1000.0 * rtb_Reset;
        (* End of Outputs for SubSystem: '<Root>/CylinderMotionControl' *)
END_CASE;

END_FUNCTION_BLOCK

// ---- StablePlatform/Function Blocks/FB_Clock.TcPOU
FUNCTION_BLOCK FB_Clock
VAR_INPUT
	bEnable 	: BOOL;
	bStart 		: BOOL;
	bStop 		: BOOL;
	fCycleTime  : LREAL;
END_VAR
VAR_OUTPUT
	fTime : LREAL;
END_VAR
VAR
END_VAR

IF bStart AND NOT(bStop) AND bEnable THEN
	fTime := fTime + fCycleTime;
ELSE
	fTime := 0.0;
END_IF

END_FUNCTION_BLOCK

// ---- StablePlatform/Function Blocks/FB_RampMotionGenerator.TcPOU
FUNCTION_BLOCK FB_RampMotionGenerator
VAR_INPUT
	bEnable: BOOL;
	bFullPeriode: BOOL;
	fCylPos0_m: LREAL;
	fCylVel0_ms: LREAL;
	fPositionSP_m: LREAL;
	fVelocitySP_ms: LREAL;
	ft0_s: LREAL;
	ftRamp_s: LREAL;
	ftHoldPos_s: LREAL;
	fSimulationTime_s: LREAL;
END_VAR
VAR_OUTPUT
	VelocityRef_ms: LREAL;
	PositionRef_m: LREAL;
END_VAR
VAR
	Error: DINT;
	slopeExt: LREAL;
	slopeRetr: LREAL;
	tHold: LREAL;
	x1: LREAL;
	x2: LREAL;
	x4: LREAL;
	x2_tmp: LREAL;
	x2_tmp_tmp: LREAL;
	x4_tmp: LREAL;
	x4_tmp_tmp: LREAL;
	x1_tmp_tmp: LREAL;
END_VAR


(* Outputs for Atomic SubSystem: '<Root>/FB_RampMotionGenerator' *)
(* MATLAB Function: '<S1>/RampSignal' *)
(* MATLAB Function 'FB_RampMotionGenerator/RampSignal': '<S2>:1' *)
(* '<S2>:1:2' x_SP = x_ref - x0; *)
(* '<S2>:1:3' vs=v_ref; *)
(* '<S2>:1:4' slopeExt=v0-vs; *)
slopeExt := fCylVel0_ms - fVelocitySP_ms;
(* '<S2>:1:5' slopeRetr=-vs-v0; *)
slopeRetr := ( -fVelocitySP_ms) - fCylVel0_ms;
(* '<S2>:1:7' as = vs/tRamp; *)
(* '<S2>:1:8' s_acc=(vs^2-v0^2)/as; *)
(* '<S2>:1:10' tHold=(x_SP-s_acc)/vs; *)
tHold := ((fPositionSP_m - fCylPos0_m) - (((fVelocitySP_ms * fVelocitySP_ms) - (fCylVel0_ms * fCylVel0_ms)) / (fVelocitySP_ms / ftRamp_s))) / fVelocitySP_ms;
(* '<S2>:1:12' if tHold < 0 *)

//IF (ABS(tHold)) < ftRamp_s THEN 
    (* '<S2>:1:13' Error = 1; *)
//    Error := 1;
//ELSE 
    (* '<S2>:1:14' else *)
    (* '<S2>:1:15' Error = 0; *)
//    Error := 0;
//END_IF;

Error := 0;

(* '<S2>:1:18' t1=tRamp; *)
(* '<S2>:1:19' t2=tHold; *)
(* '<S2>:1:20' t3=tRamp; *)
(* '<S2>:1:21' t4=tWait; *)
(* '<S2>:1:22' t5=t1; *)
(* '<S2>:1:23' t6=t2; *)
(* '<S2>:1:24' t7=t3; *)
(* '<S2>:1:26' x1 = x0 + v0*((t0+t1)-t0)-(slopeExt/t1)*((t0+t1)-t0)^2/2; *)
x2_tmp_tmp := ft0_s + ftRamp_s;
x2_tmp := x2_tmp_tmp - ft0_s;
x1_tmp_tmp := slopeExt / ftRamp_s;
x1 := ((x2_tmp * fCylVel0_ms) + fCylPos0_m) - ((x1_tmp_tmp * (x2_tmp * x2_tmp)) / 2.0);
(* '<S2>:1:27' x2 = x1 + vs*((t0+t1+t2)-(t0+t1)); *)
x2_tmp := x2_tmp_tmp + tHold;
x2 := ((x2_tmp - x2_tmp_tmp) * fVelocitySP_ms) + x1;
(* '<S2>:1:28' x4 = x_ref - v0*((t0+t1+t2+t3+t4+t5)-(t0+t1+t2+t3+t4))+(slopeRetr/t5)*((t0+t1+t2+t3+t4+t5)-(t0+t1+t2+t3+t4))^2/2; *)
x4_tmp_tmp := x2_tmp + ftRamp_s;
x4_tmp := x4_tmp_tmp + ftHoldPos_s;
x4 := (x4_tmp + ftRamp_s) - x4_tmp;
x4 := (fPositionSP_m - (x4 * fCylVel0_ms)) + (((slopeRetr / ftRamp_s) * (x4 * x4)) / 2.0);
(* '<S2>:1:29' x5 = x4-vs*((t0+t1+t2+t3+t4+t5+t6)-(t0+t1+t2+t3+t4+t5)); *)
(* '<S2>:1:31' if FullPeriode == 1 *)

IF bFullPeriode THEN 
    (* '<S2>:1:32' if Error == 1 *)

